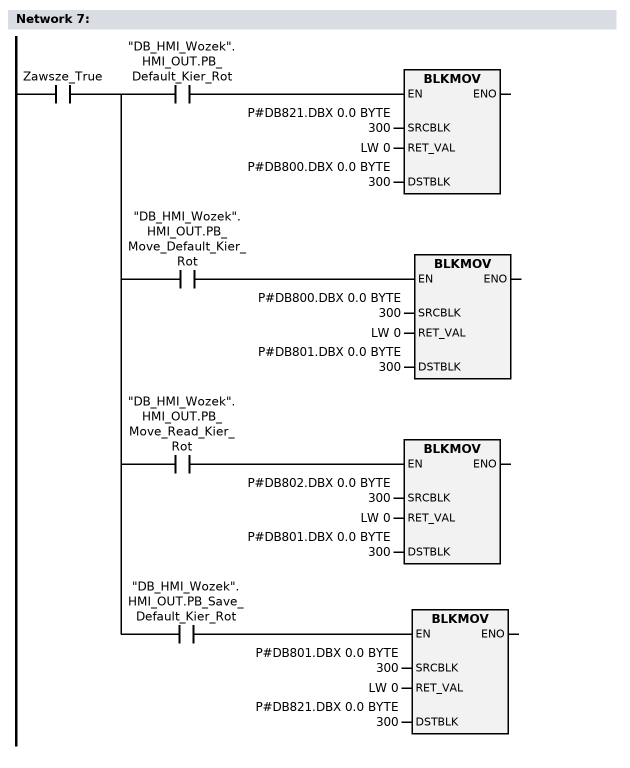
NETWORK
TITLE =
      A     "Zawsze_True";
      =     L 2.0;
      A     L 2.0;
      A     "DB_HMI_Wozek".HMI_OUT.PB_Default_Kier_Rot;
      JNB   _001;
      CALL  "BLKMOV" (
           SRCBLK                   := P#DB821.DBX 0.0 BYTE 300,
           RET_VAL                  := LW 0,
           DSTBLK                   := P#DB800.DBX 0.0 BYTE 300);
_001: NOP   0;
      A     L 2.0;
      A     "DB_HMI_Wozek".HMI_OUT.PB_Move_Default_Kier_Rot;
      JNB   _002;
      CALL  "BLKMOV" (
           SRCBLK                   := P#DB800.DBX 0.0 BYTE 300,
           RET_VAL                  := LW 0,
           DSTBLK                   := P#DB801.DBX 0.0 BYTE 300);
_002: NOP   0;
      A     L 2.0;
      A     "DB_HMI_Wozek".HMI_OUT.PB_Move_Read_Kier_Rot;
      JNB   _003;
      CALL  "BLKMOV" (
           SRCBLK                   := P#DB802.DBX 0.0 BYTE 300,
           RET_VAL                  := LW 0,
           DSTBLK                   := P#DB801.DBX 0.0 BYTE 300);
_003: NOP   0;
      A     L 2.0;
      A     "DB_HMI_Wozek".HMI_OUT.PB_Save_Default_Kier_Rot;
      JNB   _004;
      CALL  "BLKMOV" (
           SRCBLK                   := P#DB801.DBX 0.0 BYTE 300,
           RET_VAL                  := LW 0,
           DSTBLK                   := P#DB821.DBX 0.0 BYTE 300);
_004: NOP   0;
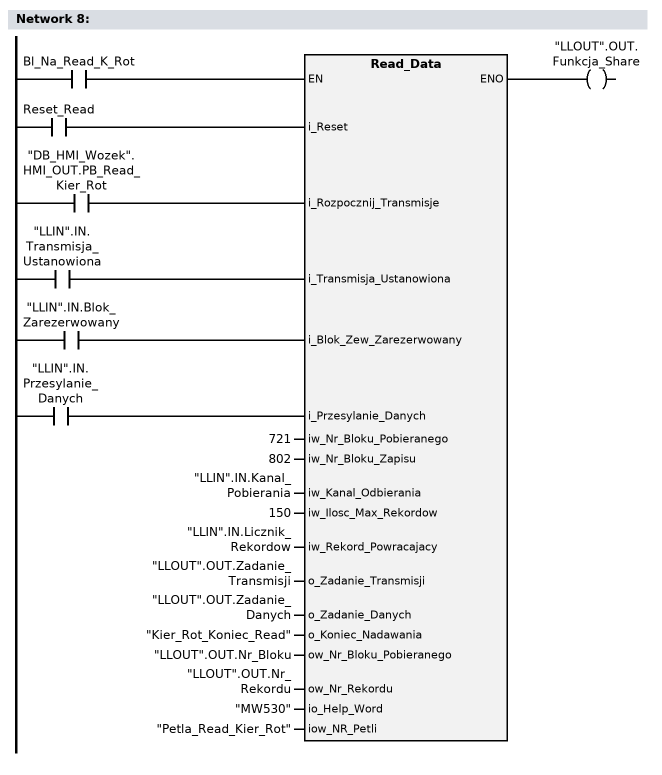
NETWORK
TITLE =
//Funkcja poboru danych
//
      A     "Reset_Read";
      =     L 2.0;
      BLD   103;
      A     "DB_HMI_Wozek".HMI_OUT.PB_Read_Kier_Rot;
      =     L 2.1;
      BLD   103;
      A     "LLIN".IN.Transmisja_Ustanowiona;
      =     L 2.2;
      BLD   103;
      A     "LLIN".IN.Blok_Zarezerwowany;
      =     L 2.3;
      BLD   103;
      A     "LLIN".IN.Przesylanie_Danych;
      =     L 2.4;
      BLD   103;
      A     "Bl_Na_Read_K_Rot";
      JNB   _005;
      CALL  "Read_Data" (
           i_Reset                  := L 2.0,
           i_Rozpocznij_Transmisje  := L 2.1,
           i_Transmisja_Ustanowiona := L 2.2,
           i_Blok_Zew_Zarezerwowany := L 2.3,
           i_Przesylanie_Danych     := L 2.4,
           iw_Nr_Bloku_Pobieranego  := 721,
           iw_Nr_Bloku_Zapisu       := 802,
           iw_Kanal_Odbierania      := "LLIN".IN.Kanal_Pobierania,
           iw_Ilosc_Max_Rekordow    := 150,
           iw_Rekord_Powracajacy    := "LLIN".IN.Licznik_Rekordow,
           o_Zadanie_Transmisji     := "LLOUT".OUT.Zadanie_Transmisji,
           o_Zadanie_Danych         := "LLOUT".OUT.Zadanie_Danych,
           o_Koniec_Nadawania       := "Kier_Rot_Koniec_Read",
           ow_Nr_Bloku_Pobieranego  := "LLOUT".OUT.Nr_Bloku,
           ow_Nr_Rekordu            := "LLOUT".OUT.Nr_Rekordu,
           io_Help_Word             := "MW530",
           iow_NR_Petli             := "Petla_Read_Kier_Rot");
_005: A     BR;
      =     "LLOUT".OUT.Funkcja_Share;
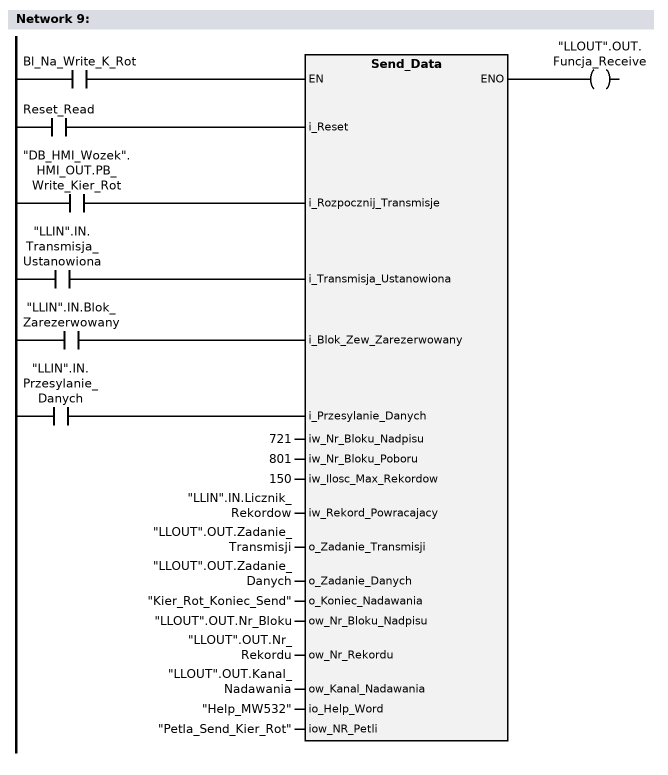
NETWORK
TITLE =
      A     "Reset_Read";
      =     L 2.0;
      BLD   103;
      A     "DB_HMI_Wozek".HMI_OUT.PB_Write_Kier_Rot;
      =     L 2.1;
      BLD   103;
      A     "LLIN".IN.Transmisja_Ustanowiona;
      =     L 2.2;
      BLD   103;
      A     "LLIN".IN.Blok_Zarezerwowany;
      =     L 2.3;
      BLD   103;
      A     "LLIN".IN.Przesylanie_Danych;
      =     L 2.4;
      BLD   103;
      A     "Bl_Na_Write_K_Rot";
      JNB   _006;
      CALL  "Send_Data" (
           i_Reset                  := L 2.0,
           i_Rozpocznij_Transmisje  := L 2.1,
           i_Transmisja_Ustanowiona := L 2.2,
           i_Blok_Zew_Zarezerwowany := L 2.3,
           i_Przesylanie_Danych     := L 2.4,
           iw_Nr_Bloku_Nadpisu      := 721,
           iw_Nr_Bloku_Poboru       := 801,
           iw_Ilosc_Max_Rekordow    := 150,
           iw_Rekord_Powracajacy    := "LLIN".IN.Licznik_Rekordow,
           o_Zadanie_Transmisji     := "LLOUT".OUT.Zadanie_Transmisji,
           o_Zadanie_Danych         := "LLOUT".OUT.Zadanie_Danych,
           o_Koniec_Nadawania       := "Kier_Rot_Koniec_Send",
           ow_Nr_Bloku_Nadpisu      := "LLOUT".OUT.Nr_Bloku,
           ow_Nr_Rekordu            := "LLOUT".OUT.Nr_Rekordu,
           ow_Kanal_Nadawania       := "LLOUT".OUT.Kanal_Nadawania,
           io_Help_Word             := "Help_MW532",
           iow_NR_Petli             := "Petla_Send_Kier_Rot");
_006: A     BR;
      =     "LLOUT".OUT.Funcja_Receive;
END_FUNCTION

FUNCTION "Ekran_Para_Odbieranie" : VOID	// FC 1730
//Ekran para odbieranie marki 505
//
VERSION : 0.1
VAR_INPUT
  Ekran_Aktywny : BOOL ;
  Timmer_Opoz : TIMER ;
END_VAR
VAR_OUTPUT
  Aktywne_Read : BOOL ;
  Aktywne_Write : BOOL ;
  Aktywna_Funkcja : BOOL ;
END_VAR
BEGIN
NETWORK
TITLE =
//Ten network celowo jest wolny
//inputy to i160
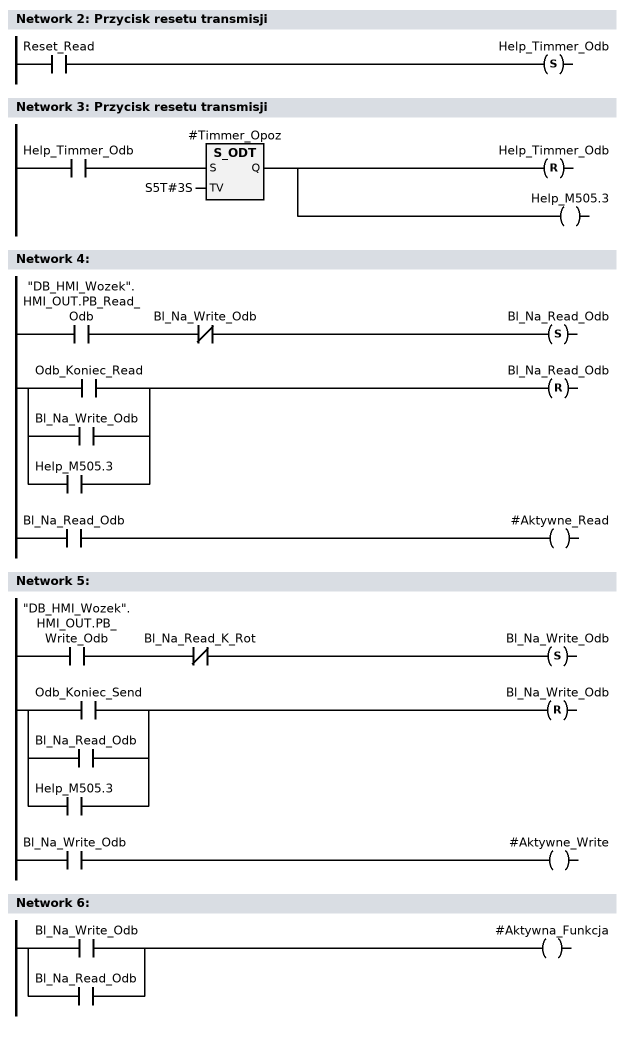
NETWORK
TITLE = Przycisk resetu transmisji
      A     "Reset_Read";
      S     "Help_Timmer_Odb";
NETWORK
TITLE = Przycisk resetu transmisji
      A     "Help_Timmer_Odb";
      L     S5T#3S;
      SD    #Timmer_Opoz;
      NOP   0;
      NOP   0;
      NOP   0;
      A     #Timmer_Opoz;
      R     "Help_Timmer_Odb";
      =     "Help_M505.3";
NETWORK
TITLE =
//Blokada NA Read
      A     "DB_HMI_Wozek".HMI_OUT.PB_Read_Odb;
      AN    "Bl_Na_Write_Odb";
      S     "Bl_Na_Read_Odb";
      A(;
      O     "Odb_Koniec_Read";
      O     "Bl_Na_Write_Odb";
      O     "Help_M505.3";
      );
      R     "Bl_Na_Read_Odb";
      A     "Bl_Na_Read_Odb";
      =     #Aktywne_Read;
NETWORK
TITLE =
//Blokada NA write
      A     "DB_HMI_Wozek".HMI_OUT.PB_Write_Odb;
      AN    "Bl_Na_Read_K_Rot";
      S     "Bl_Na_Write_Odb";
      A(;
      O     "Odb_Koniec_Send";
      O     "Bl_Na_Read_Odb";
      O     "Help_M505.3";
      );
      R     "Bl_Na_Write_Odb";
      A     "Bl_Na_Write_Odb";
      =     #Aktywne_Write;
NETWORK
TITLE =
      O     "Bl_Na_Write_Odb";
      O     "Bl_Na_Read_Odb";
      =     #Aktywna_Funkcja;
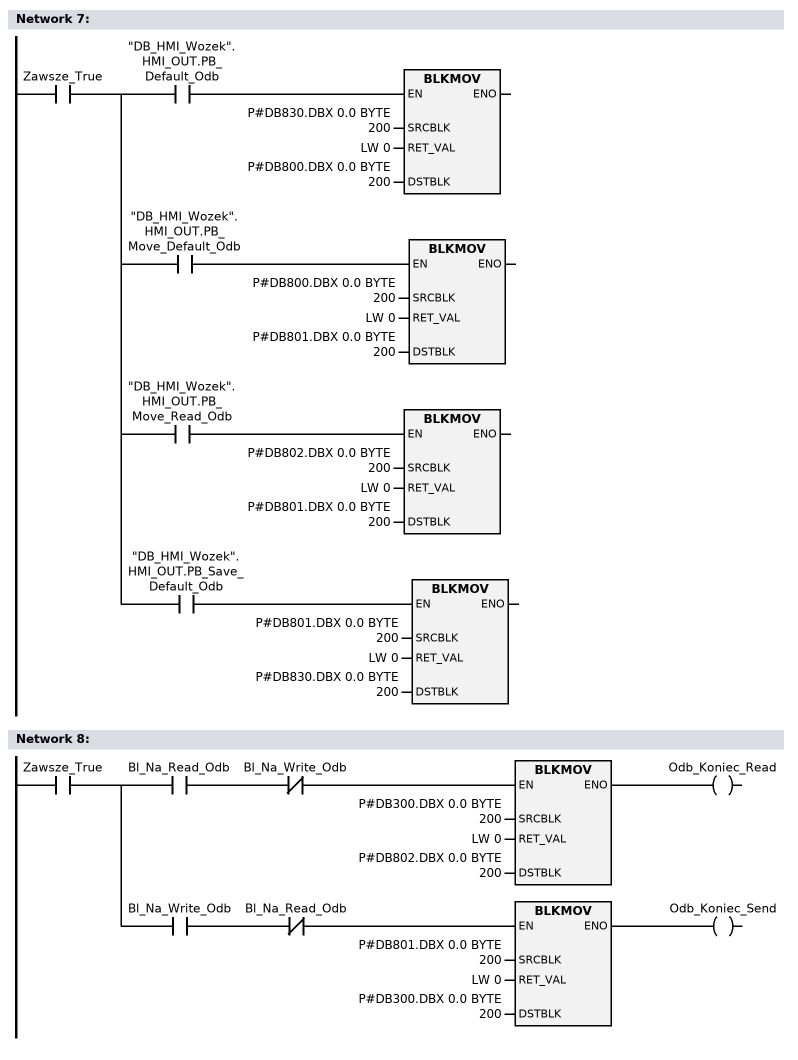
NETWORK
TITLE =
      A     "Zawsze_True";
      =     L 2.0;
      A     L 2.0;
      A     "DB_HMI_Wozek".HMI_OUT.PB_Default_Odb;
      JNB   _001;
      CALL  "BLKMOV" (
           SRCBLK                   := P#DB830.DBX 0.0 BYTE 200,
           RET_VAL                  := LW 0,
           DSTBLK                   := P#DB800.DBX 0.0 BYTE 200);
_001: NOP   0;
      A     L 2.0;
      A     "DB_HMI_Wozek".HMI_OUT.PB_Move_Default_Odb;
      JNB   _002;
      CALL  "BLKMOV" (
           SRCBLK                   := P#DB800.DBX 0.0 BYTE 200,
           RET_VAL                  := LW 0,
           DSTBLK                   := P#DB801.DBX 0.0 BYTE 200);
_002: NOP   0;
      A     L 2.0;
      A     "DB_HMI_Wozek".HMI_OUT.PB_Move_Read_Odb;
      JNB   _003;
      CALL  "BLKMOV" (
           SRCBLK                   := P#DB802.DBX 0.0 BYTE 200,
           RET_VAL                  := LW 0,
           DSTBLK                   := P#DB801.DBX 0.0 BYTE 200);
_003: NOP   0;
      A     L 2.0;
      A     "DB_HMI_Wozek".HMI_OUT.PB_Save_Default_Odb;
      JNB   _004;
      CALL  "BLKMOV" (
           SRCBLK                   := P#DB801.DBX 0.0 BYTE 200,
           RET_VAL                  := LW 0,
           DSTBLK                   := P#DB830.DBX 0.0 BYTE 200);
_004: NOP   0;
NETWORK
TITLE =
//Przesuwanie danych do bloku 300
      A     "Zawsze_True";
      =     L 2.0;
      A     L 2.0;
      A     "Bl_Na_Read_Odb";
      AN    "Bl_Na_Write_Odb";
      JNB   _005;
      CALL  "BLKMOV" (
           SRCBLK                   := P#DB300.DBX 0.0 BYTE 200,
           RET_VAL                  := LW 0,
           DSTBLK                   := P#DB802.DBX 0.0 BYTE 200);
_005: A     BR;
      =     "Odb_Koniec_Read";
      A     L 2.0;
      A     "Bl_Na_Write_Odb";
      AN    "Bl_Na_Read_Odb";
      JNB   _006;
      CALL  "BLKMOV" (
           SRCBLK                   := P#DB801.DBX 0.0 BYTE 200,
           RET_VAL                  := LW 0,
           DSTBLK                   := P#DB300.DBX 0.0 BYTE 200);
_006: A     BR;
      =     "Odb_Koniec_Send";
END_FUNCTION

DATA_BLOCK "Instancja_FB1"	// DB 1
AUTHOR : Kng
VERSION : 0.0
"Stan_Shuttle"
BEGIN
END_DATA_BLOCK

DATA_BLOCK "Instancja_FB3"	// DB 3
AUTHOR : Kng
VERSION : 0.0
"Stanowisko_KB1"
BEGIN
END_DATA_BLOCK

DATA_BLOCK "Instancja_FB4"	// DB 4
AUTHOR : Kng
VERSION : 0.0
"Stanowisko_KB2"
BEGIN
END_DATA_BLOCK

DATA_BLOCK DB 5
VERSION : 0.0
"FB_Uzbrajanie"
BEGIN
END_DATA_BLOCK

DATA_BLOCK DB 6
VERSION : 0.0
"Stan_Intro_Odbieranie"
BEGIN
END_DATA_BLOCK

DATA_BLOCK DB 7
VERSION : 0.0
"Stan_Intro_Pob_I1"
BEGIN
END_DATA_BLOCK

DATA_BLOCK DB 8
AUTHOR : Kng
VERSION : 0.0
"Stan_Intro_Pob_I2"
BEGIN
END_DATA_BLOCK

DATA_BLOCK DB 9
VERSION : 0.0
"Stan_Intro_Pob_I3"
BEGIN
END_DATA_BLOCK

DATA_BLOCK "DB_CONECTOR_KB1"	// DB 11
AUTHOR : Kng
NAME : KB1
VERSION : 0.1
  STRUCT
   Banda_Segbert : UDT 1;	//Adres 1 (Wirtualny)
   Tasma_Obrotnica : UDT 1;	//Adres 2
   Winda : UDT 1;	//Adres 3
   Banda_Wylot_2 : UDT 1;	//Adres 4
   Shuttle : UDT 1;	//Adres 5 (Wirtualny)
   Obrotnica_Pelna : UDT 6;	//Adres 9 (Wirtualny)
   Czujniki_Obr : UDT 7;	//Adres 10
   EStop_Pulpit : UDT 3;	//Adres 20
   Estop_Grzyb_Bezp : UDT 3;	//Adres 21
   Estop_Shuttle : UDT 3;	//ADres 22
  END_STRUCT ;	
BEGIN
   Obrotnica_Pelna.Silnik_OK := TRUE;
END_DATA_BLOCK

DATA_BLOCK "DB_CONECTOR_KB2"	// DB 12
AUTHOR : Kng
NAME : KB2
VERSION : 0.1
  STRUCT
   Banda_Segbert : UDT 1;	//Adres 1 (Wirtualny)
   Tasma_Obrotnica : UDT 1;	//Adres 2
   Winda : UDT 1;	//Adres 3
   Banda_Wylot_2 : UDT 1;	//Adres 4
   Shuttle : UDT 1;	//Adres 5 (Wirtualny)
   Obrotnica_Pelna : UDT 6;	//Adres 9 (Wirtualny)
   Czujniki_Obr : UDT 7;	//Adres 10
   EStop_Pulpit : UDT 3;	//Adres 20
   Estop_Grzyb_Bezp : UDT 3;	//Adres 21
   Estop_Shuttle : UDT 3;	//ADres 22
  END_STRUCT ;	
BEGIN
   Obrotnica_Pelna.Silnik_OK := TRUE;
END_DATA_BLOCK

DATA_BLOCK "DB_CONNECTOR_BUFF"	// DB 13
AUTHOR : Kng
NAME : Buff
VERSION : 0.1
  STRUCT
   Banda_2 : UDT 1;	//Temporary placeholder variable
   Banda_3 : UDT 1;
   Banda_4 : UDT 1;
   Banda_5 : UDT 1;
   Banda_6 : UDT 1;
   Banda_Rez : UDT 1;
   Banda_12 : UDT 1;
   banda_13 : UDT 1;
   Banda_14 : UDT 1;
   Banda_15 : UDT 1;
   Banda_16 : UDT 1;
   Not_Aus_1 : UDT 3;
   Not_Aus_2 : UDT 3;
   Banda_O1_Shuttle : UDT 1;
   Banda_I1_Shuttle : UDT 1;
   Banda_7 : UDT 1;
   Banda_8 : UDT 1;
   Banda_17 : UDT 1;
   Banda_18 : UDT 1;
   Not_Aus_3 : UDT 3;
   Banda_I2_Shuttle : UDT 1;
   Banda_I3_Shuttle : UDT 1;
  END_STRUCT ;	
BEGIN
END_DATA_BLOCK

DATA_BLOCK "DB_CONNECTOR_GEN"	// DB 14
AUTHOR : Kng
NAME : GENDER
VERSION : 0.1
  STRUCT
   Banda_0_Shuttle : UDT 1;	//Adres 1 (Wirtualny)
   Banda_1_Gender : UDT 1;	//Adres 2 (Wirtualny)
  END_STRUCT ;	
BEGIN
END_DATA_BLOCK

DATA_BLOCK "DB_ASI_Prosty_Odczyt_KB1"	// DB 82
AUTHOR : Kng
NAME : KB1
VERSION : 0.1
  STRUCT
   Adres_1_bit_0 : BOOL ;	//Temporary placeholder variable
   Adres_1_bit_1 : BOOL ;
   Adres_1_bit_2 : BOOL ;
   Adres_1_bit_3 : BOOL ;
   Adres_0_bit_0 : BOOL ;	//Temporary placeholder variable
   Adres_0_bit_1 : BOOL ;
   Adres_0_bit_2 : BOOL ;
   Adres_0_bit_3 : BOOL ;
   Adres_3_bit_0 : BOOL ;	//Temporary placeholder variable
   Adres_3_bit_1 : BOOL ;
   Adres_3_bit_2 : BOOL ;
   Adres_3_bit_3 : BOOL ;
   Adres_2_bit_0 : BOOL ;	//Temporary placeholder variable
   Adres_2_bit_1 : BOOL ;
   Adres_2_bit_2 : BOOL ;
   Adres_2_bit_3 : BOOL ;
   Adres_5_bit_0 : BOOL ;	//Temporary placeholder variable
   Adres_5_bit_1 : BOOL ;
   Adres_5_bit_2 : BOOL ;
   Adres_5_bit_3 : BOOL ;
   Adres_4_bit_0 : BOOL ;	//Temporary placeholder variable
   Adres_4_bit_1 : BOOL ;
   Adres_4_bit_2 : BOOL ;
   Adres_4_bit_3 : BOOL ;
   Adres_7_bit_0 : BOOL ;	//Temporary placeholder variable
   Adres_7_bit_1 : BOOL ;
   Adres_7_bit_2 : BOOL ;
   Adres_7_bit_3 : BOOL ;
   Adres_6_bit_0 : BOOL ;	//Temporary placeholder variable
   Adres_6_bit_1 : BOOL ;
   Adres_6_bit_2 : BOOL ;
   Adres_6_bit_3 : BOOL ;
   Adres_9_bit_0 : BOOL ;	//Temporary placeholder variable
   Adres_9_bit_1 : BOOL ;
   Adres_9_bit_2 : BOOL ;
   Adres_9_bit_3 : BOOL ;
   Adres_8_bit_0 : BOOL ;	//Temporary placeholder variable
   Adres_8_bit_1 : BOOL ;
   Adres_8_bit_2 : BOOL ;
   Adres_8_bit_3 : BOOL ;
   Adres_11_bit_0 : BOOL ;	//Temporary placeholder variable
   Adres_11_bit_1 : BOOL ;
   Adres_11_bit_2 : BOOL ;
   Adres_11_bit_3 : BOOL ;
   Adres_10_bit_0 : BOOL ;	//Temporary placeholder variable
   Adres_10_bit_1 : BOOL ;
   Adres_10_bit_2 : BOOL ;
   Adres_10_bit_3 : BOOL ;
   Adres_13_bit_0 : BOOL ;	//Temporary placeholder variable
   Adres_13_bit_1 : BOOL ;
   Adres_13_bit_2 : BOOL ;
   Adres_13_bit_3 : BOOL ;
   Adres_12_bit_0 : BOOL ;	//Temporary placeholder variable
   Adres_12_bit_1 : BOOL ;
   Adres_12_bit_2 : BOOL ;
   Adres_12_bit_3 : BOOL ;
   Adres_15_bit_0 : BOOL ;	//Temporary placeholder variable
   Adres_15_bit_1 : BOOL ;
   Adres_15_bit_2 : BOOL ;
   Adres_15_bit_3 : BOOL ;
   Adres_14_bit_0 : BOOL ;	//Temporary placeholder variable
   Adres_14_bit_1 : BOOL ;
   Adres_14_bit_2 : BOOL ;
   Adres_14_bit_3 : BOOL ;
   Adres_17_bit_0 : BOOL ;	//Temporary placeholder variable
   Adres_17_bit_1 : BOOL ;
   Adres_17_bit_2 : BOOL ;
   Adres_17_bit_3 : BOOL ;
   Adres_16_bit_0 : BOOL ;	//Temporary placeholder variable
   Adres_16_bit_1 : BOOL ;
   Adres_16_bit_2 : BOOL ;
   Adres_16_bit_3 : BOOL ;
   Adres_19_bit_0 : BOOL ;	//Temporary placeholder variable
   Adres_19_bit_1 : BOOL ;
   Adres_19_bit_2 : BOOL ;
   Adres_19_bit_3 : BOOL ;
   Adres_18_bit_0 : BOOL ;	//Temporary placeholder variable
   Adres_18_bit_1 : BOOL ;
   Adres_18_bit_2 : BOOL ;
   Adres_18_bit_3 : BOOL ;
   Adres_21_bit_0 : BOOL ;	//Temporary placeholder variable
   Adres_21_bit_1 : BOOL ;
   Adres_21_bit_2 : BOOL ;
   Adres_21_bit_3 : BOOL ;
   Adres_20_bit_0 : BOOL ;	//Temporary placeholder variable
   Adres_20_bit_1 : BOOL ;
   Adres_20_bit_2 : BOOL ;
   Adres_20_bit_3 : BOOL ;
   Adres_23_bit_0 : BOOL ;	//Temporary placeholder variable
   Adres_23_bit_1 : BOOL ;
   Adres_23_bit_2 : BOOL ;
   Adres_23_bit_3 : BOOL ;
   Adres_22_bit_0 : BOOL ;	//Temporary placeholder variable
   Adres_22_bit_1 : BOOL ;
   Adres_22_bit_2 : BOOL ;
   Adres_22_bit_3 : BOOL ;
   Adres_25_bit_0 : BOOL ;	//Temporary placeholder variable
   Adres_25_bit_1 : BOOL ;
   Adres_25_bit_2 : BOOL ;
   Adres_25_bit_3 : BOOL ;
   Adres_24_bit_0 : BOOL ;	//Temporary placeholder variable
   Adres_24_bit_1 : BOOL ;
   Adres_24_bit_2 : BOOL ;
   Adres_24_bit_3 : BOOL ;
   Adres_27_bit_0 : BOOL ;	//Temporary placeholder variable
   Adres_27_bit_1 : BOOL ;
   Adres_27_bit_2 : BOOL ;
   Adres_27_bit_3 : BOOL ;
   Adres_26_bit_0 : BOOL ;	//Temporary placeholder variable
   Adres_26_bit_1 : BOOL ;
   Adres_26_bit_2 : BOOL ;
   Adres_26_bit_3 : BOOL ;
   Adres_29_bit_0 : BOOL ;	//Temporary placeholder variable
   Adres_29_bit_1 : BOOL ;
   Adres_29_bit_2 : BOOL ;
   Adres_29_bit_3 : BOOL ;
   Adres_28_bit_0 : BOOL ;	//Temporary placeholder variable
   Adres_28_bit_1 : BOOL ;
   Adres_28_bit_2 : BOOL ;
   Adres_28_bit_3 : BOOL ;
   Adres_31_bit_0 : BOOL ;	//Temporary placeholder variable
   Adres_31_bit_1 : BOOL ;
   Adres_31_bit_2 : BOOL ;
   Adres_31_bit_3 : BOOL ;
   Adres_30_bit_0 : BOOL ;	//Temporary placeholder variable
   Adres_30_bit_1 : BOOL ;
   Adres_30_bit_2 : BOOL ;
   Adres_30_bit_3 : BOOL ;
  END_STRUCT ;	
BEGIN
END_DATA_BLOCK

DATA_BLOCK "DB_ASI_Prosty_Zapis_KB1"	// DB 83
AUTHOR : Kng
NAME : KB1
VERSION : 0.1
  STRUCT
   Adres_1_bit_0 : BOOL ;	//Temporary placeholder variable
   Adres_1_bit_1 : BOOL ;
   Adres_1_bit_2 : BOOL ;
   Adres_1_bit_3 : BOOL ;
   Adres_0_bit_0 : BOOL ;	//Temporary placeholder variable
   Adres_0_bit_1 : BOOL ;
   Adres_0_bit_2 : BOOL ;
   Adres_0_bit_3 : BOOL ;
   Adres_3_bit_0 : BOOL ;	//Temporary placeholder variable
   Adres_3_bit_1 : BOOL ;
   Adres_3_bit_2 : BOOL ;
   Adres_3_bit_3 : BOOL ;
   Adres_2_bit_0 : BOOL ;	//Temporary placeholder variable
   Adres_2_bit_1 : BOOL ;
   Adres_2_bit_2 : BOOL ;
   Adres_2_bit_3 : BOOL ;
   Adres_5_bit_0 : BOOL ;	//Temporary placeholder variable
   Adres_5_bit_1 : BOOL ;
   Adres_5_bit_2 : BOOL ;
   Adres_5_bit_3 : BOOL ;
   Adres_4_bit_0 : BOOL ;	//Temporary placeholder variable
   Adres_4_bit_1 : BOOL ;
   Adres_4_bit_2 : BOOL ;
   Adres_4_bit_3 : BOOL ;
   Adres_7_bit_0 : BOOL ;	//Temporary placeholder variable
   Adres_7_bit_1 : BOOL ;
   Adres_7_bit_2 : BOOL ;
   Adres_7_bit_3 : BOOL ;
   Adres_6_bit_0 : BOOL ;	//Temporary placeholder variable
   Adres_6_bit_1 : BOOL ;
   Adres_6_bit_2 : BOOL ;
   Adres_6_bit_3 : BOOL ;
   Adres_9_bit_0 : BOOL ;	//Temporary placeholder variable
   Adres_9_bit_1 : BOOL ;
   Adres_9_bit_2 : BOOL ;
   Adres_9_bit_3 : BOOL ;
   Adres_8_bit_0 : BOOL ;	//Temporary placeholder variable
   Adres_8_bit_1 : BOOL ;
   Adres_8_bit_2 : BOOL ;
   Adres_8_bit_3 : BOOL ;
   Adres_11_bit_0 : BOOL ;	//Temporary placeholder variable
   Adres_11_bit_1 : BOOL ;
   Adres_11_bit_2 : BOOL ;
   Adres_11_bit_3 : BOOL ;
   Adres_10_bit_0 : BOOL ;	//Temporary placeholder variable
   Adres_10_bit_1 : BOOL ;
   Adres_10_bit_2 : BOOL ;
   Adres_10_bit_3 : BOOL ;
   Adres_13_bit_0 : BOOL ;	//Temporary placeholder variable
   Adres_13_bit_1 : BOOL ;
   Adres_13_bit_2 : BOOL ;
   Adres_13_bit_3 : BOOL ;
   Adres_12_bit_0 : BOOL ;	//Temporary placeholder variable
   Adres_12_bit_1 : BOOL ;
   Adres_12_bit_2 : BOOL ;
   Adres_12_bit_3 : BOOL ;
   Adres_15_bit_0 : BOOL ;	//Temporary placeholder variable
   Adres_15_bit_1 : BOOL ;
   Adres_15_bit_2 : BOOL ;
   Adres_15_bit_3 : BOOL ;
   Adres_14_bit_0 : BOOL ;	//Temporary placeholder variable
   Adres_14_bit_1 : BOOL ;
   Adres_14_bit_2 : BOOL ;
   Adres_14_bit_3 : BOOL ;
   Adres_17_bit_0 : BOOL ;	//Temporary placeholder variable
   Adres_17_bit_1 : BOOL ;
   Adres_17_bit_2 : BOOL ;
   Adres_17_bit_3 : BOOL ;
   Adres_16_bit_0 : BOOL ;	//Temporary placeholder variable
   Adres_16_bit_1 : BOOL ;
   Adres_16_bit_2 : BOOL ;
   Adres_16_bit_3 : BOOL ;
   Adres_19_bit_0 : BOOL ;	//Temporary placeholder variable
   Adres_19_bit_1 : BOOL ;
   Adres_19_bit_2 : BOOL ;
   Adres_19_bit_3 : BOOL ;
   Adres_18_bit_0 : BOOL ;	//Temporary placeholder variable
   Adres_18_bit_1 : BOOL ;
   Adres_18_bit_2 : BOOL ;
   Adres_18_bit_3 : BOOL ;
   Adres_21_bit_0 : BOOL ;	//Temporary placeholder variable
   Adres_21_bit_1 : BOOL ;
   Adres_21_bit_2 : BOOL ;
   Adres_21_bit_3 : BOOL ;
   Adres_20_bit_0 : BOOL ;	//Temporary placeholder variable
   Adres_20_bit_1 : BOOL ;
   Adres_20_bit_2 : BOOL ;
   Adres_20_bit_3 : BOOL ;
   Adres_23_bit_0 : BOOL ;	//Temporary placeholder variable
   Adres_23_bit_1 : BOOL ;
   Adres_23_bit_2 : BOOL ;
   Adres_23_bit_3 : BOOL ;
   Adres_22_bit_0 : BOOL ;	//Temporary placeholder variable
   Adres_22_bit_1 : BOOL ;
   Adres_22_bit_2 : BOOL ;
   Adres_22_bit_3 : BOOL ;
   Adres_25_bit_0 : BOOL ;	//Temporary placeholder variable
   Adres_25_bit_1 : BOOL ;
   Adres_25_bit_2 : BOOL ;
   Adres_25_bit_3 : BOOL ;
   Adres_24_bit_0 : BOOL ;	//Temporary placeholder variable
   Adres_24_bit_1 : BOOL ;
   Adres_24_bit_2 : BOOL ;
   Adres_24_bit_3 : BOOL ;
   Adres_27_bit_0 : BOOL ;	//Temporary placeholder variable
   Adres_27_bit_1 : BOOL ;
   Adres_27_bit_2 : BOOL ;
   Adres_27_bit_3 : BOOL ;
   Adres_26_bit_0 : BOOL ;	//Temporary placeholder variable
   Adres_26_bit_1 : BOOL ;
   Adres_26_bit_2 : BOOL ;
   Adres_26_bit_3 : BOOL ;
   Adres_29_bit_0 : BOOL ;	//Temporary placeholder variable
   Adres_29_bit_1 : BOOL ;
   Adres_29_bit_2 : BOOL ;
   Adres_29_bit_3 : BOOL ;
   Adres_28_bit_0 : BOOL ;	//Temporary placeholder variable
   Adres_28_bit_1 : BOOL ;
   Adres_28_bit_2 : BOOL ;
   Adres_28_bit_3 : BOOL ;
   Adres_31_bit_0 : BOOL ;	//Temporary placeholder variable
   Adres_31_bit_1 : BOOL ;
   Adres_31_bit_2 : BOOL ;
   Adres_31_bit_3 : BOOL ;
   Adres_30_bit_0 : BOOL ;	//Temporary placeholder variable
   Adres_30_bit_1 : BOOL ;
   Adres_30_bit_2 : BOOL ;
   Adres_30_bit_3 : BOOL ;
  END_STRUCT ;	
BEGIN
END_DATA_BLOCK

DATA_BLOCK "DB_ASI_Prosty_Odczyt_KB2"	// DB 84
AUTHOR : Kng
NAME : KB2
VERSION : 0.1
  STRUCT
   Adres_1_bit_0 : BOOL ;	//Temporary placeholder variable
   Adres_1_bit_1 : BOOL ;
   Adres_1_bit_2 : BOOL ;
   Adres_1_bit_3 : BOOL ;
   Adres_0_bit_0 : BOOL ;	//Temporary placeholder variable
   Adres_0_bit_1 : BOOL ;
   Adres_0_bit_2 : BOOL ;
   Adres_0_bit_3 : BOOL ;
   Adres_3_bit_0 : BOOL ;	//Temporary placeholder variable
   Adres_3_bit_1 : BOOL ;
   Adres_3_bit_2 : BOOL ;
   Adres_3_bit_3 : BOOL ;
   Adres_2_bit_0 : BOOL ;	//Temporary placeholder variable
   Adres_2_bit_1 : BOOL ;
   Adres_2_bit_2 : BOOL ;
   Adres_2_bit_3 : BOOL ;
   Adres_5_bit_0 : BOOL ;	//Temporary placeholder variable
   Adres_5_bit_1 : BOOL ;
   Adres_5_bit_2 : BOOL ;
   Adres_5_bit_3 : BOOL ;
   Adres_4_bit_0 : BOOL ;	//Temporary placeholder variable
   Adres_4_bit_1 : BOOL ;
   Adres_4_bit_2 : BOOL ;
   Adres_4_bit_3 : BOOL ;
   Adres_7_bit_0 : BOOL ;	//Temporary placeholder variable
   Adres_7_bit_1 : BOOL ;
   Adres_7_bit_2 : BOOL ;
   Adres_7_bit_3 : BOOL ;
   Adres_6_bit_0 : BOOL ;	//Temporary placeholder variable
   Adres_6_bit_1 : BOOL ;
   Adres_6_bit_2 : BOOL ;
   Adres_6_bit_3 : BOOL ;
   Adres_9_bit_0 : BOOL ;	//Temporary placeholder variable
   Adres_9_bit_1 : BOOL ;
   Adres_9_bit_2 : BOOL ;
   Adres_9_bit_3 : BOOL ;
   Adres_8_bit_0 : BOOL ;	//Temporary placeholder variable
   Adres_8_bit_1 : BOOL ;
   Adres_8_bit_2 : BOOL ;
   Adres_8_bit_3 : BOOL ;
   Adres_11_bit_0 : BOOL ;	//Temporary placeholder variable
   Adres_11_bit_1 : BOOL ;
   Adres_11_bit_2 : BOOL ;
   Adres_11_bit_3 : BOOL ;
   Adres_10_bit_0 : BOOL ;	//Temporary placeholder variable
   Adres_10_bit_1 : BOOL ;
   Adres_10_bit_2 : BOOL ;
   Adres_10_bit_3 : BOOL ;
   Adres_13_bit_0 : BOOL ;	//Temporary placeholder variable
   Adres_13_bit_1 : BOOL ;
   Adres_13_bit_2 : BOOL ;
   Adres_13_bit_3 : BOOL ;
   Adres_12_bit_0 : BOOL ;	//Temporary placeholder variable
   Adres_12_bit_1 : BOOL ;
   Adres_12_bit_2 : BOOL ;
   Adres_12_bit_3 : BOOL ;
   Adres_15_bit_0 : BOOL ;	//Temporary placeholder variable
   Adres_15_bit_1 : BOOL ;
   Adres_15_bit_2 : BOOL ;
   Adres_15_bit_3 : BOOL ;
   Adres_14_bit_0 : BOOL ;	//Temporary placeholder variable
   Adres_14_bit_1 : BOOL ;
   Adres_14_bit_2 : BOOL ;
   Adres_14_bit_3 : BOOL ;
   Adres_17_bit_0 : BOOL ;	//Temporary placeholder variable
   Adres_17_bit_1 : BOOL ;
   Adres_17_bit_2 : BOOL ;
   Adres_17_bit_3 : BOOL ;
   Adres_16_bit_0 : BOOL ;	//Temporary placeholder variable
   Adres_16_bit_1 : BOOL ;
   Adres_16_bit_2 : BOOL ;
   Adres_16_bit_3 : BOOL ;
   Adres_19_bit_0 : BOOL ;	//Temporary placeholder variable
   Adres_19_bit_1 : BOOL ;
   Adres_19_bit_2 : BOOL ;
   Adres_19_bit_3 : BOOL ;
   Adres_18_bit_0 : BOOL ;	//Temporary placeholder variable
   Adres_18_bit_1 : BOOL ;
   Adres_18_bit_2 : BOOL ;
   Adres_18_bit_3 : BOOL ;
   Adres_21_bit_0 : BOOL ;	//Temporary placeholder variable
   Adres_21_bit_1 : BOOL ;
   Adres_21_bit_2 : BOOL ;
   Adres_21_bit_3 : BOOL ;
   Adres_20_bit_0 : BOOL ;	//Temporary placeholder variable
   Adres_20_bit_1 : BOOL ;
   Adres_20_bit_2 : BOOL ;
   Adres_20_bit_3 : BOOL ;
   Adres_23_bit_0 : BOOL ;	//Temporary placeholder variable
   Adres_23_bit_1 : BOOL ;
   Adres_23_bit_2 : BOOL ;
   Adres_23_bit_3 : BOOL ;
   Adres_22_bit_0 : BOOL ;	//Temporary placeholder variable
   Adres_22_bit_1 : BOOL ;
   Adres_22_bit_2 : BOOL ;
   Adres_22_bit_3 : BOOL ;
   Adres_25_bit_0 : BOOL ;	//Temporary placeholder variable
   Adres_25_bit_1 : BOOL ;
   Adres_25_bit_2 : BOOL ;
   Adres_25_bit_3 : BOOL ;
   Adres_24_bit_0 : BOOL ;	//Temporary placeholder variable
   Adres_24_bit_1 : BOOL ;
   Adres_24_bit_2 : BOOL ;
   Adres_24_bit_3 : BOOL ;
   Adres_27_bit_0 : BOOL ;	//Temporary placeholder variable
   Adres_27_bit_1 : BOOL ;
   Adres_27_bit_2 : BOOL ;
   Adres_27_bit_3 : BOOL ;
   Adres_26_bit_0 : BOOL ;	//Temporary placeholder variable
   Adres_26_bit_1 : BOOL ;
   Adres_26_bit_2 : BOOL ;
   Adres_26_bit_3 : BOOL ;
   Adres_29_bit_0 : BOOL ;	//Temporary placeholder variable
   Adres_29_bit_1 : BOOL ;
   Adres_29_bit_2 : BOOL ;
   Adres_29_bit_3 : BOOL ;
   Adres_28_bit_0 : BOOL ;	//Temporary placeholder variable
   Adres_28_bit_1 : BOOL ;
   Adres_28_bit_2 : BOOL ;
   Adres_28_bit_3 : BOOL ;
   Adres_31_bit_0 : BOOL ;	//Temporary placeholder variable
   Adres_31_bit_1 : BOOL ;
   Adres_31_bit_2 : BOOL ;
   Adres_31_bit_3 : BOOL ;
   Adres_30_bit_0 : BOOL ;	//Temporary placeholder variable
   Adres_30_bit_1 : BOOL ;
   Adres_30_bit_2 : BOOL ;
   Adres_30_bit_3 : BOOL ;
  END_STRUCT ;	
BEGIN
END_DATA_BLOCK

DATA_BLOCK "DB_ASi_Prosty_Zapis_KB2"	// DB 85
AUTHOR : Kng
NAME : KB2
VERSION : 0.1
  STRUCT
   Adres_1_bit_0 : BOOL ;	//Temporary placeholder variable
   Adres_1_bit_1 : BOOL ;
   Adres_1_bit_2 : BOOL ;
   Adres_1_bit_3 : BOOL ;
   Adres_0_bit_0 : BOOL ;	//Temporary placeholder variable
   Adres_0_bit_1 : BOOL ;
   Adres_0_bit_2 : BOOL ;
   Adres_0_bit_3 : BOOL ;
   Adres_3_bit_0 : BOOL ;	//Temporary placeholder variable
   Adres_3_bit_1 : BOOL ;
   Adres_3_bit_2 : BOOL ;
   Adres_3_bit_3 : BOOL ;
   Adres_2_bit_0 : BOOL ;	//Temporary placeholder variable
   Adres_2_bit_1 : BOOL ;
   Adres_2_bit_2 : BOOL ;
   Adres_2_bit_3 : BOOL ;
   Adres_5_bit_0 : BOOL ;	//Temporary placeholder variable
   Adres_5_bit_1 : BOOL ;
   Adres_5_bit_2 : BOOL ;
   Adres_5_bit_3 : BOOL ;
   Adres_4_bit_0 : BOOL ;	//Temporary placeholder variable
   Adres_4_bit_1 : BOOL ;
   Adres_4_bit_2 : BOOL ;
   Adres_4_bit_3 : BOOL ;
   Adres_7_bit_0 : BOOL ;	//Temporary placeholder variable
   Adres_7_bit_1 : BOOL ;
   Adres_7_bit_2 : BOOL ;
   Adres_7_bit_3 : BOOL ;
   Adres_6_bit_0 : BOOL ;	//Temporary placeholder variable
   Adres_6_bit_1 : BOOL ;
   Adres_6_bit_2 : BOOL ;
   Adres_6_bit_3 : BOOL ;
   Adres_9_bit_0 : BOOL ;	//Temporary placeholder variable
   Adres_9_bit_1 : BOOL ;
   Adres_9_bit_2 : BOOL ;
   Adres_9_bit_3 : BOOL ;
   Adres_8_bit_0 : BOOL ;	//Temporary placeholder variable
   Adres_8_bit_1 : BOOL ;
   Adres_8_bit_2 : BOOL ;
   Adres_8_bit_3 : BOOL ;
   Adres_11_bit_0 : BOOL ;	//Temporary placeholder variable
   Adres_11_bit_1 : BOOL ;
   Adres_11_bit_2 : BOOL ;
   Adres_11_bit_3 : BOOL ;
   Adres_10_bit_0 : BOOL ;	//Temporary placeholder variable
   Adres_10_bit_1 : BOOL ;
   Adres_10_bit_2 : BOOL ;
   Adres_10_bit_3 : BOOL ;
   Adres_13_bit_0 : BOOL ;	//Temporary placeholder variable
   Adres_13_bit_1 : BOOL ;
   Adres_13_bit_2 : BOOL ;
   Adres_13_bit_3 : BOOL ;
   Adres_12_bit_0 : BOOL ;	//Temporary placeholder variable
   Adres_12_bit_1 : BOOL ;
   Adres_12_bit_2 : BOOL ;
   Adres_12_bit_3 : BOOL ;
   Adres_15_bit_0 : BOOL ;	//Temporary placeholder variable
   Adres_15_bit_1 : BOOL ;
   Adres_15_bit_2 : BOOL ;
   Adres_15_bit_3 : BOOL ;
   Adres_14_bit_0 : BOOL ;	//Temporary placeholder variable
   Adres_14_bit_1 : BOOL ;
   Adres_14_bit_2 : BOOL ;
   Adres_14_bit_3 : BOOL ;
   Adres_17_bit_0 : BOOL ;	//Temporary placeholder variable
   Adres_17_bit_1 : BOOL ;
   Adres_17_bit_2 : BOOL ;
   Adres_17_bit_3 : BOOL ;
   Adres_16_bit_0 : BOOL ;	//Temporary placeholder variable
   Adres_16_bit_1 : BOOL ;
   Adres_16_bit_2 : BOOL ;
   Adres_16_bit_3 : BOOL ;
   Adres_19_bit_0 : BOOL ;	//Temporary placeholder variable
   Adres_19_bit_1 : BOOL ;
   Adres_19_bit_2 : BOOL ;
   Adres_19_bit_3 : BOOL ;
   Adres_18_bit_0 : BOOL ;	//Temporary placeholder variable
   Adres_18_bit_1 : BOOL ;
   Adres_18_bit_2 : BOOL ;
   Adres_18_bit_3 : BOOL ;
   Adres_21_bit_0 : BOOL ;	//Temporary placeholder variable
   Adres_21_bit_1 : BOOL ;
   Adres_21_bit_2 : BOOL ;
   Adres_21_bit_3 : BOOL ;
   Adres_20_bit_0 : BOOL ;	//Temporary placeholder variable
   Adres_20_bit_1 : BOOL ;
   Adres_20_bit_2 : BOOL ;
   Adres_20_bit_3 : BOOL ;
   Adres_23_bit_0 : BOOL ;	//Temporary placeholder variable
   Adres_23_bit_1 : BOOL ;
   Adres_23_bit_2 : BOOL ;
   Adres_23_bit_3 : BOOL ;
   Adres_22_bit_0 : BOOL ;	//Temporary placeholder variable
   Adres_22_bit_1 : BOOL ;
   Adres_22_bit_2 : BOOL ;
   Adres_22_bit_3 : BOOL ;
   Adres_25_bit_0 : BOOL ;	//Temporary placeholder variable
   Adres_25_bit_1 : BOOL ;
   Adres_25_bit_2 : BOOL ;
   Adres_25_bit_3 : BOOL ;
   Adres_24_bit_0 : BOOL ;	//Temporary placeholder variable
   Adres_24_bit_1 : BOOL ;
   Adres_24_bit_2 : BOOL ;
   Adres_24_bit_3 : BOOL ;
   Adres_27_bit_0 : BOOL ;	//Temporary placeholder variable
   Adres_27_bit_1 : BOOL ;
   Adres_27_bit_2 : BOOL ;
   Adres_27_bit_3 : BOOL ;
   Adres_26_bit_0 : BOOL ;	//Temporary placeholder variable
   Adres_26_bit_1 : BOOL ;
   Adres_26_bit_2 : BOOL ;
   Adres_26_bit_3 : BOOL ;
   Adres_29_bit_0 : BOOL ;	//Temporary placeholder variable
   Adres_29_bit_1 : BOOL ;
   Adres_29_bit_2 : BOOL ;
   Adres_29_bit_3 : BOOL ;
   Adres_28_bit_0 : BOOL ;	//Temporary placeholder variable
   Adres_28_bit_1 : BOOL ;
   Adres_28_bit_2 : BOOL ;
   Adres_28_bit_3 : BOOL ;
   Adres_31_bit_0 : BOOL ;	//Temporary placeholder variable
   Adres_31_bit_1 : BOOL ;
   Adres_31_bit_2 : BOOL ;
   Adres_31_bit_3 : BOOL ;
   Adres_30_bit_0 : BOOL ;	//Temporary placeholder variable
   Adres_30_bit_1 : BOOL ;
   Adres_30_bit_2 : BOOL ;
   Adres_30_bit_3 : BOOL ;
  END_STRUCT ;	
BEGIN
END_DATA_BLOCK

DATA_BLOCK "DB_ASi_Prosty_Odczyt_Buf"	// DB 86
AUTHOR : Kng
NAME : Buff
VERSION : 0.1
  STRUCT
   Adres_1_bit_0 : BOOL ;	//Temporary placeholder variable
   Adres_1_bit_1 : BOOL ;
   Adres_1_bit_2 : BOOL ;
   Adres_1_bit_3 : BOOL ;
   Adres_0_bit_0 : BOOL ;	//Temporary placeholder variable
   Adres_0_bit_1 : BOOL ;
   Adres_0_bit_2 : BOOL ;
   Adres_0_bit_3 : BOOL ;
   Adres_3_bit_0 : BOOL ;	//Temporary placeholder variable
   Adres_3_bit_1 : BOOL ;
   Adres_3_bit_2 : BOOL ;
   Adres_3_bit_3 : BOOL ;
   Adres_2_bit_0 : BOOL ;	//Temporary placeholder variable
   Adres_2_bit_1 : BOOL ;
   Adres_2_bit_2 : BOOL ;
   Adres_2_bit_3 : BOOL ;
   Adres_5_bit_0 : BOOL ;	//Temporary placeholder variable
   Adres_5_bit_1 : BOOL ;
   Adres_5_bit_2 : BOOL ;
   Adres_5_bit_3 : BOOL ;
   Adres_4_bit_0 : BOOL ;	//Temporary placeholder variable
   Adres_4_bit_1 : BOOL ;
   Adres_4_bit_2 : BOOL ;
   Adres_4_bit_3 : BOOL ;
   Adres_7_bit_0 : BOOL ;	//Temporary placeholder variable
   Adres_7_bit_1 : BOOL ;
   Adres_7_bit_2 : BOOL ;
   Adres_7_bit_3 : BOOL ;
   Adres_6_bit_0 : BOOL ;	//Temporary placeholder variable
   Adres_6_bit_1 : BOOL ;
   Adres_6_bit_2 : BOOL ;
   Adres_6_bit_3 : BOOL ;
   Adres_9_bit_0 : BOOL ;	//Temporary placeholder variable
   Adres_9_bit_1 : BOOL ;
   Adres_9_bit_2 : BOOL ;
   Adres_9_bit_3 : BOOL ;
   Adres_8_bit_0 : BOOL ;	//Temporary placeholder variable
   Adres_8_bit_1 : BOOL ;
   Adres_8_bit_2 : BOOL ;
   Adres_8_bit_3 : BOOL ;
   Adres_11_bit_0 : BOOL ;	//Temporary placeholder variable
   Adres_11_bit_1 : BOOL ;
   Adres_11_bit_2 : BOOL ;
   Adres_11_bit_3 : BOOL ;
   Adres_10_bit_0 : BOOL ;	//Temporary placeholder variable
   Adres_10_bit_1 : BOOL ;
   Adres_10_bit_2 : BOOL ;
   Adres_10_bit_3 : BOOL ;
   Adres_13_bit_0 : BOOL ;	//Temporary placeholder variable
   Adres_13_bit_1 : BOOL ;
   Adres_13_bit_2 : BOOL ;
   Adres_13_bit_3 : BOOL ;
   Adres_12_bit_0 : BOOL ;	//Temporary placeholder variable
   Adres_12_bit_1 : BOOL ;
   Adres_12_bit_2 : BOOL ;
   Adres_12_bit_3 : BOOL ;
   Adres_15_bit_0 : BOOL ;	//Temporary placeholder variable
   Adres_15_bit_1 : BOOL ;
   Adres_15_bit_2 : BOOL ;
   Adres_15_bit_3 : BOOL ;
   Adres_14_bit_0 : BOOL ;	//Temporary placeholder variable
   Adres_14_bit_1 : BOOL ;
   Adres_14_bit_2 : BOOL ;
   Adres_14_bit_3 : BOOL ;
   Adres_17_bit_0 : BOOL ;	//Temporary placeholder variable
   Adres_17_bit_1 : BOOL ;
   Adres_17_bit_2 : BOOL ;
   Adres_17_bit_3 : BOOL ;
   Adres_16_bit_0 : BOOL ;	//Temporary placeholder variable
   Adres_16_bit_1 : BOOL ;
   Adres_16_bit_2 : BOOL ;
   Adres_16_bit_3 : BOOL ;
   Adres_19_bit_0 : BOOL ;	//Temporary placeholder variable
   Adres_19_bit_1 : BOOL ;
   Adres_19_bit_2 : BOOL ;
   Adres_19_bit_3 : BOOL ;
   Adres_18_bit_0 : BOOL ;	//Temporary placeholder variable
   Adres_18_bit_1 : BOOL ;
   Adres_18_bit_2 : BOOL ;
   Adres_18_bit_3 : BOOL ;
   Adres_21_bit_0 : BOOL ;	//Temporary placeholder variable
   Adres_21_bit_1 : BOOL ;
   Adres_21_bit_2 : BOOL ;
   Adres_21_bit_3 : BOOL ;
   Adres_20_bit_0 : BOOL ;	//Temporary placeholder variable
   Adres_20_bit_1 : BOOL ;
   Adres_20_bit_2 : BOOL ;
   Adres_20_bit_3 : BOOL ;
   Adres_23_bit_0 : BOOL ;	//Temporary placeholder variable
   Adres_23_bit_1 : BOOL ;
   Adres_23_bit_2 : BOOL ;
   Adres_23_bit_3 : BOOL ;
   Adres_22_bit_0 : BOOL ;	//Temporary placeholder variable
   Adres_22_bit_1 : BOOL ;
   Adres_22_bit_2 : BOOL ;
   Adres_22_bit_3 : BOOL ;
   Adres_25_bit_0 : BOOL ;	//Temporary placeholder variable
   Adres_25_bit_1 : BOOL ;
   Adres_25_bit_2 : BOOL ;
   Adres_25_bit_3 : BOOL ;
   Adres_24_bit_0 : BOOL ;	//Temporary placeholder variable
   Adres_24_bit_1 : BOOL ;
   Adres_24_bit_2 : BOOL ;
   Adres_24_bit_3 : BOOL ;
   Adres_27_bit_0 : BOOL ;	//Temporary placeholder variable
   Adres_27_bit_1 : BOOL ;
   Adres_27_bit_2 : BOOL ;
   Adres_27_bit_3 : BOOL ;
   Adres_26_bit_0 : BOOL ;	//Temporary placeholder variable
   Adres_26_bit_1 : BOOL ;
   Adres_26_bit_2 : BOOL ;
   Adres_26_bit_3 : BOOL ;
   Adres_29_bit_0 : BOOL ;	//Temporary placeholder variable
   Adres_29_bit_1 : BOOL ;
   Adres_29_bit_2 : BOOL ;
   Adres_29_bit_3 : BOOL ;
   Adres_28_bit_0 : BOOL ;	//Temporary placeholder variable
   Adres_28_bit_1 : BOOL ;
   Adres_28_bit_2 : BOOL ;
   Adres_28_bit_3 : BOOL ;
   Adres_31_bit_0 : BOOL ;	//Temporary placeholder variable
   Adres_31_bit_1 : BOOL ;
   Adres_31_bit_2 : BOOL ;
   Adres_31_bit_3 : BOOL ;
   Adres_30_bit_0 : BOOL ;	//Temporary placeholder variable
   Adres_30_bit_1 : BOOL ;
   Adres_30_bit_2 : BOOL ;
   Adres_30_bit_3 : BOOL ;
  END_STRUCT ;	
BEGIN
END_DATA_BLOCK

DATA_BLOCK "DB_ASi_Prosty_Zapis_Buf"	// DB 87
AUTHOR : Kng
NAME : Buff
VERSION : 0.1
  STRUCT
   Adres_1_bit_0 : BOOL ;	//Temporary placeholder variable
   Adres_1_bit_1 : BOOL ;
   Adres_1_bit_2 : BOOL ;
   Adres_1_bit_3 : BOOL ;
   Adres_0_bit_0 : BOOL ;	//Temporary placeholder variable
   Adres_0_bit_1 : BOOL ;
   Adres_0_bit_2 : BOOL ;
   Adres_0_bit_3 : BOOL ;
   Adres_3_bit_0 : BOOL ;	//Temporary placeholder variable
   Adres_3_bit_1 : BOOL ;
   Adres_3_bit_2 : BOOL ;
   Adres_3_bit_3 : BOOL ;
   Adres_2_bit_0 : BOOL ;	//Temporary placeholder variable
   Adres_2_bit_1 : BOOL ;
   Adres_2_bit_2 : BOOL ;
   Adres_2_bit_3 : BOOL ;
   Adres_5_bit_0 : BOOL ;	//Temporary placeholder variable
   Adres_5_bit_1 : BOOL ;
   Adres_5_bit_2 : BOOL ;
   Adres_5_bit_3 : BOOL ;
   Adres_4_bit_0 : BOOL ;	//Temporary placeholder variable
   Adres_4_bit_1 : BOOL ;
   Adres_4_bit_2 : BOOL ;
   Adres_4_bit_3 : BOOL ;
   Adres_7_bit_0 : BOOL ;	//Temporary placeholder variable
   Adres_7_bit_1 : BOOL ;
   Adres_7_bit_2 : BOOL ;
   Adres_7_bit_3 : BOOL ;
   Adres_6_bit_0 : BOOL ;	//Temporary placeholder variable
   Adres_6_bit_1 : BOOL ;
   Adres_6_bit_2 : BOOL ;
   Adres_6_bit_3 : BOOL ;
   Adres_9_bit_0 : BOOL ;	//Temporary placeholder variable
   Adres_9_bit_1 : BOOL ;
   Adres_9_bit_2 : BOOL ;
   Adres_9_bit_3 : BOOL ;
   Adres_8_bit_0 : BOOL ;	//Temporary placeholder variable
   Adres_8_bit_1 : BOOL ;
   Adres_8_bit_2 : BOOL ;
   Adres_8_bit_3 : BOOL ;
   Adres_11_bit_0 : BOOL ;	//Temporary placeholder variable
   Adres_11_bit_1 : BOOL ;
   Adres_11_bit_2 : BOOL ;
   Adres_11_bit_3 : BOOL ;
   Adres_10_bit_0 : BOOL ;	//Temporary placeholder variable
   Adres_10_bit_1 : BOOL ;
   Adres_10_bit_2 : BOOL ;
   Adres_10_bit_3 : BOOL ;
   Adres_13_bit_0 : BOOL ;	//Temporary placeholder variable
   Adres_13_bit_1 : BOOL ;
   Adres_13_bit_2 : BOOL ;
   Adres_13_bit_3 : BOOL ;
   Adres_12_bit_0 : BOOL ;	//Temporary placeholder variable
   Adres_12_bit_1 : BOOL ;
   Adres_12_bit_2 : BOOL ;
   Adres_12_bit_3 : BOOL ;
   Adres_15_bit_0 : BOOL ;	//Temporary placeholder variable
   Adres_15_bit_1 : BOOL ;
   Adres_15_bit_2 : BOOL ;
   Adres_15_bit_3 : BOOL ;
   Adres_14_bit_0 : BOOL ;	//Temporary placeholder variable
   Adres_14_bit_1 : BOOL ;
   Adres_14_bit_2 : BOOL ;
   Adres_14_bit_3 : BOOL ;
   Adres_17_bit_0 : BOOL ;	//Temporary placeholder variable
   Adres_17_bit_1 : BOOL ;
   Adres_17_bit_2 : BOOL ;
   Adres_17_bit_3 : BOOL ;
   Adres_16_bit_0 : BOOL ;	//Temporary placeholder variable
   Adres_16_bit_1 : BOOL ;
   Adres_16_bit_2 : BOOL ;
   Adres_16_bit_3 : BOOL ;
   Adres_19_bit_0 : BOOL ;	//Temporary placeholder variable
   Adres_19_bit_1 : BOOL ;
   Adres_19_bit_2 : BOOL ;
   Adres_19_bit_3 : BOOL ;
   Adres_18_bit_0 : BOOL ;	//Temporary placeholder variable
   Adres_18_bit_1 : BOOL ;
   Adres_18_bit_2 : BOOL ;
   Adres_18_bit_3 : BOOL ;
   Adres_21_bit_0 : BOOL ;	//Temporary placeholder variable
   Adres_21_bit_1 : BOOL ;
   Adres_21_bit_2 : BOOL ;
   Adres_21_bit_3 : BOOL ;
   Adres_20_bit_0 : BOOL ;	//Temporary placeholder variable
   Adres_20_bit_1 : BOOL ;
   Adres_20_bit_2 : BOOL ;
   Adres_20_bit_3 : BOOL ;
   Adres_23_bit_0 : BOOL ;	//Temporary placeholder variable
   Adres_23_bit_1 : BOOL ;
   Adres_23_bit_2 : BOOL ;
   Adres_23_bit_3 : BOOL ;
   Adres_22_bit_0 : BOOL ;	//Temporary placeholder variable
   Adres_22_bit_1 : BOOL ;
   Adres_22_bit_2 : BOOL ;
   Adres_22_bit_3 : BOOL ;
   Adres_25_bit_0 : BOOL ;	//Temporary placeholder variable
   Adres_25_bit_1 : BOOL ;
   Adres_25_bit_2 : BOOL ;
   Adres_25_bit_3 : BOOL ;
   Adres_24_bit_0 : BOOL ;	//Temporary placeholder variable
   Adres_24_bit_1 : BOOL ;
   Adres_24_bit_2 : BOOL ;
   Adres_24_bit_3 : BOOL ;
   Adres_27_bit_0 : BOOL ;	//Temporary placeholder variable
   Adres_27_bit_1 : BOOL ;
   Adres_27_bit_2 : BOOL ;
   Adres_27_bit_3 : BOOL ;
   Adres_26_bit_0 : BOOL ;	//Temporary placeholder variable
   Adres_26_bit_1 : BOOL ;
   Adres_26_bit_2 : BOOL ;
   Adres_26_bit_3 : BOOL ;
   Adres_29_bit_0 : BOOL ;	//Temporary placeholder variable
   Adres_29_bit_1 : BOOL ;
   Adres_29_bit_2 : BOOL ;
   Adres_29_bit_3 : BOOL ;
   Adres_28_bit_0 : BOOL ;	//Temporary placeholder variable
   Adres_28_bit_1 : BOOL ;
   Adres_28_bit_2 : BOOL ;
   Adres_28_bit_3 : BOOL ;
   Adres_31_bit_0 : BOOL ;	//Temporary placeholder variable
   Adres_31_bit_1 : BOOL ;
   Adres_31_bit_2 : BOOL ;
   Adres_31_bit_3 : BOOL ;
   Adres_30_bit_0 : BOOL ;	//Temporary placeholder variable
   Adres_30_bit_1 : BOOL ;
   Adres_30_bit_2 : BOOL ;
   Adres_30_bit_3 : BOOL ;
  END_STRUCT ;	
BEGIN
END_DATA_BLOCK

DATA_BLOCK "Bledy_Shuttle"	// DB 116
VERSION : 0.1
  STRUCT
   Bledy : STRUCT
    Przek_Bezp_Nie_Ok : BOOL ;	//Blad przekanika bezpieczenstwa [I4.1 s. 10]
    Blad_Kom_Odbieranie : BOOL ;	//Blad komunikacji z odbieraniem [FC119]
    Bezpieczniki_Nie_Ok : BOOL ;	//Wyzwolenie wylacznika termicznego [I4.0 s. 10]
    Mayser_Nie_Ok : BOOL ;	//Wyzwolenie listwy bezpieczenstwa [I4.2 s.10]
    Foto_Zle_Pokrycie : BOOL ;	//Niedozwolone pokrycie fotokomorek obecnosci palety [I5.2,I5.3 s.11]
    Hamulec_Reczny_Rewizja : BOOL ;	//Hamulec reczny odbezpieczony [I5.6 s 11]
    Skaner_Wym_Przod_Reset : BOOL ;	//Skaner przod wymagany reset [I6.1 s.12]
    Skaner_Przod_Error : BOOL ;	//Blad Skanera przedniego lub jego  zabrudzenie [I6.2 s.12]
    Skaner_Przod_Strefa : BOOL ;	//Skaner przedni strefa wyzwolona I[I6.3 s.12]
    Skaner_Wym_Tyl_Reset : BOOL ;	//Skaner tylni wymagany reset [I7.1 s.12]
    Skaner_Tyl_Error : BOOL ;	//Blad Skanera tylniego lub jego  zabrudzenie [I7.2 s.12]
    Skaner_Tyl_Strefa : BOOL ;	//Skaner tylni strefa wyzwolona [I7.3 s.12]
    Obwody_Zew_Nie_Ok : BOOL ;	//Obwody bezpieczenstwa zewnetrzne nie Ok [I8.1 s.14](Not-Aus Slupy)
    Falownik_Sew_Blad : BOOL ;	//Blad falownika SEW [FC101]
    Falownik_Sew_N_Ready : BOOL ;	//Falownik sew nie gotowy [FC101]
    Falownik_Lenze_Blad : BOOL ;	//Blad falownika Lenze [FC101]
    Warunki_Startu_N_OK : BOOL ;	//Warunki startu Sew nie spelnione [FC101]
    Blad_Zwolnienia : BOOL ;	//Blad zwolnienia tasmy transportera [FC30]
    Help_int : INT ;	//Rezerwa dla booli
    Nr_Bledu_Sew : INT ;	//Blad specyficzny sew do odczytania
    Prad_Aktualny : INT ;	//Prad aktualny SEW [FC101]
    Predkosc_Aktualna : INT ;	//Predkosc akutualna wozka [FC101]
    Reserwa_Int : INT ;
    REserwa_Int1 : INT ;
   END_STRUCT ;
  END_STRUCT ;	
BEGIN
END_DATA_BLOCK

DATA_BLOCK "Bledy_KB1"	// DB 117
VERSION : 0.1
  STRUCT
   Obwod_Bezp_1_Nie_OK : BOOL ;	//Przekaznik bezpieczenstwa stanowisko nie ok [I24.0-KB2]{I14.0-KB1] s.12
   Obwod_Bezp_2_Nie_OK : BOOL ;	//Przekaznik bezpieczenstwa wozek nie ok [I24.1-KB2][I14.1-KB1] s.12
   Petla_Bezp_Nie_Ok : BOOL ;	//Petla bezpiecznikow nie OK [I24.2-KB2][I14.2-KB1] s.12
   Blad_Silnika_Rolki_Obr : BOOL ;	//Blad silnika rolek obrotnica Adres 2 s.32
   Blad_Silnika_Rolki_Winda : BOOL ;	//Blad silnika rolek winda Adres 3 s.33
   Blad_Silnika_Rolki_Wy_2 : BOOL ;	//Blad silnika rolek wylot 2 Adres 4 s.34
   Blad_Silnika_Obrotu : BOOL ;	//Blad falownika Lenze obronicy Adres DP [8-KB2][4-KB1] s.35
   Blad_Not_Aus_Pulpit : BOOL ;	//Przycisk Not-Aus pulpit sterowniczy Adres 20 s.40
   Blad_Not_Aus_Grzyb_Obr : BOOL ;	//Blad Not-Aus grzyb obrotnica Adres 21 s.40
   Blad_Not_Aus_Wozek : BOOL ;	//Blad Not-Aus na s³upie od wozka Adres 22 s.40
  END_STRUCT ;	
BEGIN
END_DATA_BLOCK

DATA_BLOCK "Bledy_KB2"	// DB 118
VERSION : 0.1
  STRUCT
   Obwod_Bezp_1_Nie_OK : BOOL ;	//Przekaznik bezpieczenstwa stanowisko nie ok [I24.0-KB2]{I14.0-KB1] s.12
   Obwod_Bezp_2_Nie_OK : BOOL ;	//Przekaznik bezpieczenstwa wozek nie ok [I24.1-KB2][I14.1-KB1] s.12
   Petla_Bezp_Nie_Ok : BOOL ;	//Petla bezpiecznikow nie OK [I24.2-KB2][I14.2-KB1] s.12
   Blad_Silnika_Rolki_Obr : BOOL ;	//Blad silnika rolek obrotnica Adres 2 s.32
   Blad_Silnika_Rolki_Winda : BOOL ;	//Blad silnika rolek winda Adres 3 s.33
   Blad_Silnika_Rolki_Wy_2 : BOOL ;	//Blad silnika rolek wylot 2 Adres 4 s.34
   Blad_Silnika_Obrotu : BOOL ;	//Blad falownika Lenze obronicy Adres DP [8-KB2][4-KB1] s.35
   Blad_Not_Aus_Pulpit : BOOL ;	//Przycisk Not-Aus pulpit sterowniczy Adres 20 s.40
   Blad_Not_Aus_Grzyb_Obr : BOOL ;	//Blad Not-Aus grzyb obrotnica Adres 21 s.40
   Blad_Not_Aus_Wozek : BOOL ;	//Blad Not-Aus na s³upie od wozka Adres 22 s.40
  END_STRUCT ;	
BEGIN
END_DATA_BLOCK

DATA_BLOCK "Bledy_Buffor"	// DB 119
VERSION : 0.1
  STRUCT
   Blad_Silnik_Banda_2 : BOOL ;	//Blad silnika Adres 2 - bandy odbieranie
   Blad_Silnik_Banda_3 : BOOL ;	//Blad silnika Adres 3 - bandy odbieranie
   Blad_Silnik_Banda_4 : BOOL ;	//Blad silnika Adres 4 - bandy odbieranie
   Blad_Silnik_Banda_5 : BOOL ;	//Blad silnika Adres 5 - bandy odbieranie
   Blad_Silnik_Banda_6 : BOOL ;	//Blad silnika Adres 6 - bandy odbieranie
   Blad_Silnik_Banda_Rez : BOOL ;
   Blad_Silnik_Banda_12 : BOOL ;	//Blad silnika Adres 12 - bandy pobieranie
   Blad_Silnik_Banda_13 : BOOL ;	//Blad silnika Adres 13 - bandy pobieranie
   Blad_Silnik_Banda_14 : BOOL ;	//Blad silnika Adres 14 - bandy pobieranie
   Blad_Silnik_Banda_15 : BOOL ;	//Blad silnika Adres 15 - bandy pobieranie
   Blad_Silnik_Banda_16 : BOOL ;	//Blad silnika Adres 16 - bandy pobieranie
   Blad_Not_Aus_Pulpit : BOOL ;	//Blad Not-Aus pulpit Adres 20
   Blad_Not_Aus_KB1 : BOOL ;	//Blad Not-Aus na slupie Kolbus 1 (Adres 22) s.9
   Blad_Not_Aus_KB2 : BOOL ;	//Blad Not-Aus na slupie Kolbus 2 (Adres 22) s.9
   Blad_Not_Aus_Slupy : BOOL ;	//Blad Not-Aus na ktoryms slupie  (Adres 22)
   Blad_Not_Aus_Buff : BOOL ;	//Blad Not-Aus na slupie Buffory  (Adres 23)
   Przekaznik_Bezp_1_Nie_Ok : BOOL ;	//Przekaznik Bezpieczenstwa Pulpit Nie OK [I10.0] s.12
   Przekaznik_Bezp_2_Nie_Ok : BOOL ;	//Przekanik Bezpieczenstwa od Wozka Nie OK [I10.1] s.12
   Blad_Wozka_Widl : BOOL ;	//Wozek przyslania fotokomorke [I8.7] s.10
   Napiecie_Shuttle_Wyl : BOOL ;	//Napiecie na szynoprzewod nie za³¹czone [Q8.3] s.18
   Blad_Silnik_Banda_7 : BOOL ;	//Blad silnika Adres 7- bandy pobieranie
   Blad_Silnik_Banda_17 : BOOL ;	//Blad silnika Adres 17 - bandy pobieranie
   Blad_Silnik_Banda_8 : BOOL ;	//Blad silnika Adres 8 - bandy pobieranie
   Blad_Silnik_Banda_18 : BOOL ;	//Blad silnika Adres 18 - bandy pobieranie
   Blad_Not_Aus_Pulpit_2 : BOOL ;	//Blad Not-Aus pulpit Adres 24
  END_STRUCT ;	
BEGIN
END_DATA_BLOCK

DATA_BLOCK "DB_HMI_KB1"	// DB 121
AUTHOR : Kng
NAME : HMI_KB2
VERSION : 0.1
  STRUCT
   HMI_IN : STRUCT 	//Zmienne wchodzace do HMI nie nadpisywane W HMI (100 bajtow)
    Reserwa_in : BOOL ;
    Winda_W_Dole : BOOL ;	//Winda w dole dbx0.1
    Winda_W_Gorze : BOOL ;	//Winda w gorze
    Zawor_Winda : BOOL ;
    Silnik_Winda : BOOL ;
    Foto_Winda_Przod : BOOL ;
    Foto_Winda_Tyl : BOOL ;
    Silnik_Banda_Winda_OK : BOOL ;
    Obrot_Pozycja_Na_Winde : BOOL ;
    Obrot_Pozycja_Na_Wylot_2 : BOOL ;
    Foto_Obrotnica_Przod : BOOL ;
    Foto_Obrotnica_Tyl : BOOL ;
    Silnik_Banda_Obrot_OK : BOOL ;
    Silnik_Obrot_OK : BOOL ;
    Foto_Wozek_Przod : BOOL ;
    Foto_Wozek_Tyl : BOOL ;
    Silnik_Wozek_OK : BOOL ;
    Foto_Segbert_Przod : BOOL ;
    Foto_Segbert_Tyl : BOOL ;
    Segbert_Strefa_Ok : BOOL ;
    Segbert_Silnik_Ok : BOOL ;
    Foto_Wylot_2_Przod : BOOL ;
    Foto_Wylot_2_Tyl : BOOL ;
    Wylot_2_Silnik_OK : BOOL ;
    Not_Aus_Pulpit_Ok : BOOL ;
    Not_Aus_Slupek_OK : BOOL ;
    Not_Aus_Wozek_OK : BOOL ;
    Uzbrajanie_Aktywne : BOOL ;	//dbx3.3
    Uzbrajanie_Kier_Lewo : BOOL ;
    Uzbrajanie_Kier_Prawo : BOOL ;
    Zasprzeglenie_KB1 : BOOL ;
    Rezerwa_113 : BOOL ;
    Silnik_Segbert_CW : BOOL ;
    Wybor_Kier_Spedycja : BOOL ;	//dbx4.1
    Wybor_Kier_Intro : BOOL ;
    Wybor_Wiazanie_Pop : BOOL ;
    Wybor_Wiazanie_Wzdl : BOOL ;
    Wybor_Deklowanie : BOOL ;
    Wybor_Foliowanie : BOOL ;
    Silnik_Segbert_CCW : BOOL ;
    Silnik_Obrot_Banda_CCW : BOOL ;
    Silnik_Obrot_Banda_CW : BOOL ;
    Silnik_Winda_CCW : BOOL ;
    Silnik_Winda_CW : BOOL ;
    Silnik_Wylot2_CCW : BOOL ;
    Silnik_Wylot2_CW : BOOL ;
    Silnik_Wozek_CCW : BOOL ;
    Silnik_Wozek_CW : BOOL ;
    Silnik_Segbert_Praca : BOOL ;
    Silnik_Obrot_Banda_Praca : BOOL ;
    Silnik_Winda_Praca : BOOL ;
    Silnik_Wylot2_Praca : BOOL ;
    Silnik_Wozek_Praca : BOOL ;
    Silnik_Obrotnica_CCW : BOOL ;
    Silnik_Obrotnica_CW : BOOL ;
    Obrotnica_Na_Winde : BYTE ;
    Obrotnica_Na_Wylot2 : BYTE ;
    Ruch_Banda_Segbert : BYTE ;
    Ruch_Banda_Obrotnicy : BYTE ;
    Ruch_Banda_Winda : BYTE ;
    Ruch_Banda_Wozek : BYTE ;
    Ruch_Banda_Wylot2 : BYTE ;
    Status_B_Segbert_uzbr : BOOL ;
    Status_B_Segbert_foliow : BOOL ;
    Status_B_Segbert_deklow : BOOL ;
    Status_B_Segbert_W_wzdl : BOOL ;
    Status_B_Segbert_W_poprz : BOOL ;
    Status_B_Segbert_widoczn : BOOL ;
    res : BOOL ;
    res1 : BOOL ;
    Status_B_Obr_0st_uzbr : BOOL ;
    Status_B_Obr_0st_foliow : BOOL ;
    Status_B_Obr_0st_deklow : BOOL ;
    Status_B_Obr_0st_W_wzdl : BOOL ;
    Status_B_Obr_0st_W_poprz : BOOL ;
    Status_B_Obr_0st_widoczn : BOOL ;
    res2 : BOOL ;
    res3 : BOOL ;
    Status_B_Winda_uzbr : BOOL ;
    Status_B_Winda_foliow : BOOL ;
    Status_B_Winda_deklow : BOOL ;
    Status_B_Winda_W_wzdl : BOOL ;
    Status_B_Winda_W_poprz : BOOL ;
    Status_B_Winda_widoczn : BOOL ;
    res10 : BOOL ;
    res11 : BOOL ;
    Status_B_Wozek_uzbr : BOOL ;
    Status_B_Wozek_foliow : BOOL ;
    Status_B_Wozek_deklow : BOOL ;
    Status_B_Wozek_W_wzdl : BOOL ;
    Status_B_Wozek_W_poprz : BOOL ;
    Status_B_Wozek_widoczn : BOOL ;
    res4 : BOOL ;
    res5 : BOOL ;
    Status_B_Wylot2_uzbr : BOOL ;
    Status_B_Wylot2_foliow : BOOL ;
    Status_B_Wylot2_deklow : BOOL ;
    Status_B_Wylot2_W_wzdl : BOOL ;
    Status_B_Wylot2_W_poprz : BOOL ;
    Status_B_Wylot2_widoczn : BOOL ;
    res6 : BOOL ;
    res7 : BOOL ;
    Status_B_Obr_90st_uzbr : BOOL ;
    Status_B_Obr_90st_foliow : BOOL ;
    Status_B_Obr_90st_deklow : BOOL ;
    Status_B_Obr_90st_W_wzdl : BOOL ;
    Status_B_Obr_90st_W_popr : BOOL ;
    Status_B_Obr_90st_widocz : BOOL ;
    res8 : BOOL ;
    res9 : BOOL ;
    Winda_Dol : BOOL ;
    Winda_Srodek_Dol : BOOL ;
    Winda_Srodek_Gora : BOOL ;
    Winda_Gora : BOOL ;
    Paleta_Winda_Inf_KB1 : DINT ;
    Paleta_Ruch_Pion : INT ;
    Paleta_Ruch_Poziom : INT ;
    Paleta_Winda_Inf_KB1_HMI : DINT ;
    Tablica_IN_INT : ARRAY  [1 .. 13 ] OF INT ;
    Tablica_IN_DWORD : ARRAY  [1 .. 8 ] OF DINT ;
    Aktualna_Data : DATE_AND_TIME ;
   END_STRUCT ;
   HMI_OUT : STRUCT 	//Zmienne wychodzace z HMI Nie nadpisywane w sterowniku od 100 bajta
    Tryb_Uzbrajania_Palety : BOOL ;	//Paleta bedzie uzbrajana dbx100.0
    Tryb_Pracy_Inline : BOOL ;	//Kierunek wylotu palety 1-winda 0-bok dbx100.1
    Ladunek_Na_Intro : BOOL ;
    Reserwa_11 : BOOL ;
    Reserwa_12 : BOOL ;
    Reset_Bledow : BOOL ;	//Reset bledow maszyny
    Reserwa_14 : BOOL ;
    Reserwa_15 : BOOL ;
    Reserwa_16 : BOOL ;
    Reserwa_17 : BOOL ;
    Reserwa_18 : BOOL ;
    Reserwa_19 : BOOL ;
    Reserwa_110 : BOOL ;
    Reserwa_111 : BOOL ;
    Reserwa_112 : BOOL ;
    Reserwa_113 : BOOL ;
    Wybrano_Kier_Spedycje : BOOL ;	//Jedzie na Gender ( dbx2.0)
    Wybrano_Kier_Intro : BOOL ;	//Jedzie na bandy buffory
    Wybrano_Wiaz_Pop : BOOL ;
    Wybrano_Wiaz_Wzdlu : BOOL ;	//Wybrano wiazanie wzdluzne
    Wybrano_Deklowanie : BOOL ;	//wybrano deklowanie
    Wybrano_Foliowanie : BOOL ;
    Kier_Spedycja_Aktywny : BOOL ;
    Kierunek_Intro_Aktywny : BOOL ;
    Wiazanie_Pop_Aktywne : BOOL ;
    Wiazanie_Wzdl_Aktywne : BOOL ;
    Deklowanie_Aktywne : BOOL ;
    Foliowanie_Aktywne : BOOL ;
    reserwa : BOOL ;
    reserwa1 : BOOL ;
    reserwa2 : BOOL ;
    reserwa3 : BOOL ;
    reserwa4 : INT ;	//Wartosc % predkosci z ladunkiem
    Predkosc_Cargo : INT ;	//Wartosc % predkosci z ladunkiem
    Tablica_OUT_INT : ARRAY  [1 .. 21 ] OF INT ;
    Maska_Zadania : INT ;
    Tablica_OUT_DWORD : ARRAY  [1 .. 9 ] OF DWORD ;
    Reserwa_DWORD : DWORD ;
    Aktualna_Data : DATE_AND_TIME ;
   END_STRUCT ;
   HMI_IN_OUT : STRUCT 	//Zmienne nadpisywane w sterowniku i w HMI od 200 bajta
    Reserwa_in_out : BOOL ;
    io_Reserwa : INT ;	//Rodzaj wybranego wlotu
    Predkosc_Obrotnicy : DINT  := L#20;	//dbd4
    Tablica_IN_OUT_INT : ARRAY  [1 .. 22 ] OF INT ;
    Tablica_IN_OUT_DWORD : ARRAY  [1 .. 10 ] OF DWORD ;
    Aktualna_Data : DATE_AND_TIME ;
   END_STRUCT ;
  END_STRUCT ;	
BEGIN
   HMI_IN_OUT.Predkosc_Obrotnicy := L#20;
END_DATA_BLOCK

DATA_BLOCK "DB_HMI_KB2"	// DB 122
AUTHOR : Kng
NAME : HMI_KB2
VERSION : 0.1
  STRUCT
   HMI_IN : STRUCT 	//Zmienne wchodzace do HMI nie nadpisywane W HMI (100 bajtow)
    Reserwa_in : BOOL ;
    Winda_W_Dole : BOOL ;	//Winda w dole dbx0.1
    Winda_W_Gorze : BOOL ;	//Winda w gorze
    Zawor_Winda : BOOL ;
    Silnik_Winda : BOOL ;
    Foto_Winda_Przod : BOOL ;
    Foto_Winda_Tyl : BOOL ;
    Silnik_Banda_Winda_OK : BOOL ;
    Obrot_Pozycja_Na_Winde : BOOL ;
    Obrot_Pozycja_Na_Wylot_2 : BOOL ;
    Foto_Obrotnica_Przod : BOOL ;
    Foto_Obrotnica_Tyl : BOOL ;
    Silnik_Banda_Obrot_OK : BOOL ;
    Silnik_Obrot_OK : BOOL ;
    Foto_Wozek_Przod : BOOL ;
    Foto_Wozek_Tyl : BOOL ;
    Silnik_Wozek_OK : BOOL ;
    Foto_Segbert_Przod : BOOL ;
    Foto_Segbert_Tyl : BOOL ;
    Segbert_Strefa_Ok : BOOL ;
    Segbert_Silnik_Ok : BOOL ;
    Foto_Wylot_2_Przod : BOOL ;
    Foto_Wylot_2_Tyl : BOOL ;
    Wylot_2_Silnik_OK : BOOL ;
    Not_Aus_Pulpit_Ok : BOOL ;
    Not_Aus_Slupek_OK : BOOL ;
    Not_Aus_Wozek_OK : BOOL ;
    Uzbrajanie_Aktywne : BOOL ;	//dbx3.3
    Uzbrajanie_Kier_Lewo : BOOL ;
    Uzbrajanie_Kier_Prawo : BOOL ;
    Zasprzeglenie_KB2 : BOOL ;
    Rezerwa_113 : BOOL ;
    Silnik_Segbert_CW : BOOL ;
    Wybor_Kier_Spedycja : BOOL ;	//dbx4.1
    Wybor_Kier_Intro : BOOL ;
    Wybor_Wiazanie_Pop : BOOL ;
    Wybor_Wiazanie_Wzdl : BOOL ;
    Wybor_Deklowanie : BOOL ;
    Wybor_Foliowanie : BOOL ;
    Silnik_Segbert_CCW : BOOL ;
    Silnik_Obrot_Banda_CCW : BOOL ;
    Silnik_Obrot_Banda_CW : BOOL ;
    Silnik_Winda_CCW : BOOL ;
    Silnik_Winda_CW : BOOL ;
    Silnik_Wylot2_CCW : BOOL ;
    Silnik_Wylot2_CW : BOOL ;
    Silnik_Wozek_CCW : BOOL ;
    Silnik_Wozek_CW : BOOL ;
    Silnik_Segbert_Praca : BOOL ;
    Silnik_Obrot_Banda_Praca : BOOL ;
    Silnik_Winda_Praca : BOOL ;
    Silnik_Wylot2_Praca : BOOL ;
    Silnik_Wozek_Praca : BOOL ;
    Silnik_Obrotnica_CCW : BOOL ;
    Silnik_Obrotnica_CW : BOOL ;
    Obrotnica_Na_Winde : BYTE ;
    Obrotnica_Na_Wylot2 : BYTE ;
    Ruch_Banda_Segbert : BYTE ;
    Ruch_Banda_Obrotnicy : BYTE ;
    Ruch_Banda_Winda : BYTE ;
    Ruch_Banda_Wozek : BYTE ;
    Ruch_Banda_Wylot2 : BYTE ;
    Status_B_Segbert_uzbr : BOOL ;
    Status_B_Segbert_foliow : BOOL ;
    Status_B_Segbert_deklow : BOOL ;
    Status_B_Segbert_W_wzdl : BOOL ;
    Status_B_Segbert_W_poprz : BOOL ;
    Status_B_Segbert_widoczn : BOOL ;
    res : BOOL ;
    res1 : BOOL ;
    Status_B_Obr_0st_uzbr : BOOL ;
    Status_B_Obr_0st_foliow : BOOL ;
    Status_B_Obr_0st_deklow : BOOL ;
    Status_B_Obr_0st_W_wzdl : BOOL ;
    Status_B_Obr_0st_W_poprz : BOOL ;
    Status_B_Obr_0st_widoczn : BOOL ;
    res2 : BOOL ;
    res3 : BOOL ;
    Status_B_Winda_uzbr : BOOL ;
    Status_B_Winda_foliow : BOOL ;
    Status_B_Winda_deklow : BOOL ;
    Status_B_Winda_W_wzdl : BOOL ;
    Status_B_Winda_W_poprz : BOOL ;
    Status_B_Winda_widoczn : BOOL ;
    res10 : BOOL ;
    res11 : BOOL ;
    Status_B_Wozek_uzbr : BOOL ;
    Status_B_Wozek_foliow : BOOL ;
    Status_B_Wozek_deklow : BOOL ;
    Status_B_Wozek_W_wzdl : BOOL ;
    Status_B_Wozek_W_poprz : BOOL ;
    Status_B_Wozek_widoczn : BOOL ;
    res4 : BOOL ;
    res5 : BOOL ;
    Status_B_Wylot2_uzbr : BOOL ;
    Status_B_Wylot2_foliow : BOOL ;
    Status_B_Wylot2_deklow : BOOL ;
    Status_B_Wylot2_W_wzdl : BOOL ;
    Status_B_Wylot2_W_poprz : BOOL ;
    Status_B_Wylot2_widoczn : BOOL ;
    res6 : BOOL ;
    res7 : BOOL ;
    Status_B_Obr_90st_uzbr : BOOL ;
    Status_B_Obr_90st_foliow : BOOL ;
    Status_B_Obr_90st_deklow : BOOL ;
    Status_B_Obr_90st_W_wzdl : BOOL ;
    Status_B_Obr_90st_W_popr : BOOL ;
    Status_B_Obr_90st_widocz : BOOL ;
    res8 : BOOL ;
    res9 : BOOL ;
    Winda_Dol : BOOL ;
    Winda_Srodek_Dol : BOOL ;
    Winda_Srodek_Gora : BOOL ;
    Winda_Gora : BOOL ;
    Paleta_Winda_Inf_KB2 : DINT ;
    Paleta_Ruch_Pion : INT ;
    Paleta_Ruch_Poziom : INT ;
    Paleta_Winda_Inf_KB2_HMI : DINT ;
    Tablica_IN_INT : ARRAY  [1 .. 13 ] OF INT ;
    Tablica_IN_DWORD : ARRAY  [1 .. 8 ] OF DINT ;
    Aktualna_Data : DATE_AND_TIME ;
   END_STRUCT ;
   HMI_OUT : STRUCT 	//Zmienne wychodzace z HMI Nie nadpisywane w sterowniku od 100 bajta
    Tryb_Uzbrajania_Palety : BOOL ;	//Paleta bedzie uzbrajana dbx100.0
    Tryb_Pracy_Inline : BOOL ;	//Kierunek wylotu palety 1-winda 0-bok dbx100.1
    Ladunek_Na_Intro : BOOL ;	//Reset bledow maszyny
    Reserwa_11 : BOOL ;
    Reserwa_12 : BOOL ;
    Reset_Bledow : BOOL ;	//Reset bledow maszyny
    Reserwa_14 : BOOL ;
    Reserwa_15 : BOOL ;
    Reserwa_16 : BOOL ;
    Reserwa_17 : BOOL ;
    Reserwa_18 : BOOL ;
    Reserwa_19 : BOOL ;
    Reserwa_110 : BOOL ;
    Reserwa_111 : BOOL ;
    Reserwa_112 : BOOL ;
    Reserwa_113 : BOOL ;
    Wybrano_Kier_Spedycje : BOOL ;	//Jedzie na Gender ( dbx2.0)
    Wybrano_Kier_Intro : BOOL ;	//Jedzie na bandy buffory
    Wybrano_Wiaz_Pop : BOOL ;
    Wybrano_Wiaz_Wzdlu : BOOL ;	//Wybrano wiazanie wzdluzne
    Wybrano_Deklowanie : BOOL ;	//wybrano deklowanie
    Wybrano_Foliowanie : BOOL ;
    Kier_Spedycja_Aktywny : BOOL ;
    Kierunek_Intro_Aktywny : BOOL ;
    Wiazanie_Pop_Aktywne : BOOL ;
    Wiazanie_Wzdl_Aktywne : BOOL ;
    Deklowanie_Aktywne : BOOL ;
    Foliowanie_Aktywne : BOOL ;
    reserwa : BOOL ;
    reserwa1 : BOOL ;
    reserwa2 : BOOL ;
    reserwa3 : BOOL ;
    reserwa4 : INT ;	//Wartosc % predkosci z ladunkiem
    Predkosc_Cargo : INT ;	//Wartosc % predkosci z ladunkiem
    Tablica_OUT_INT : ARRAY  [1 .. 21 ] OF INT ;
    Maska_Zadania : INT ;
    Tablica_OUT_DWORD : ARRAY  [1 .. 9 ] OF DWORD ;
    Reserwa_DWORD : DWORD ;
    Aktualna_Data : DATE_AND_TIME ;
   END_STRUCT ;
   HMI_IN_OUT : STRUCT 	//Zmienne nadpisywane w sterowniku i w HMI od 200 bajta
    Reserwa_in_out : BOOL ;
    io_Reserwa : INT ;	//Rodzaj wybranego wlotu
    Predkosc_Obrotnicy : DINT  := L#20;	//dbd4
    Tablica_IN_OUT_INT : ARRAY  [1 .. 22 ] OF INT ;
    Tablica_IN_OUT_DWORD : ARRAY  [1 .. 10 ] OF DWORD ;
    Aktualna_Data : DATE_AND_TIME ;
   END_STRUCT ;
  END_STRUCT ;	
BEGIN
   HMI_IN_OUT.Predkosc_Obrotnicy := L#20;
END_DATA_BLOCK

DATA_BLOCK "DB_HMI_BUF"	// DB 123
AUTHOR : Kng
NAME : HMI_BUFF
VERSION : 0.1
  STRUCT
   HMI_IN : STRUCT 	//Zmienne wchodzace do HMI nie nadpisywane W HMI (100 bajtow)
    Linia_Buffory_Auto : BOOL ;	//Linia buforow jest auto
    Linia_Buffory_Reczny : BOOL ;	//Linia buforow jest w recznym
    Zawsze_True : BOOL ;
    Zawsze_False : BOOL ;
    res255 : BOOL ;
    res54 : BOOL ;
    res11 : BOOL ;
    re32 : BOOL ;
    ret : BOOL ;
    rettt : BOOL ;
    zxc : BOOL ;
    fd : BOOL ;
    zz : BOOL ;
    ddd : BOOL ;
    rrr : BOOL ;
    ttt : BOOL ;
    Linia_Gender_Online : BOOL ;
    Linia_Gender_Offline : BOOL ;
    Linia_Gender_Blad : BOOL ;
    Linia_Blad_Komunikacji : BOOL ;
    Linia_Gender_Auto : BOOL ;
    Linia_Gender_Reczny : BOOL ;
    Linia_Gender_Mark_Bezp : BOOL ;
    Rezerwa_17 : BOOL ;
    Rezerwa_18 : BOOL ;
    Rezerwa_19 : BOOL ;
    Rezerwa_110 : BOOL ;
    Rezerwa_111 : BOOL ;
    Rezerwa_112 : BOOL ;
    Rezerwa_113 : BOOL ;
    Rezerwa_114 : BOOL ;
    Rezerwa_115 : BOOL ;
    Rezerwa_116 : BOOL ;
    I1_Wybor_Kier_Sped : BOOL ;
    I1_Wybor_Kier_Intro : BOOL ;
    I1_Wybor_Wiaz_Pop : BOOL ;
    I1_Wybor_Wiaz_Wzdl : BOOL ;
    I1_Wybor_Deklowanie : BOOL ;
    I1_Wybor_Foliowanie : BOOL ;
    Rezerwa_200 : BOOL ;
    Rezerwa_2001 : BOOL ;
    Rezerwa_2002 : BOOL ;
    Rezerwa_2003 : BOOL ;
    Rezerwa_2004 : BOOL ;
    Rezerwa_2005 : BOOL ;
    Rezerwa_2006 : BOOL ;
    Rezerwa_2007 : BOOL ;
    Rezerwa_2008 : BOOL ;
    rezerwa2009 : BOOL ;
    I2_Wybor_Kier_Sped : BOOL ;
    I2_Wybor_Kier_Intro : BOOL ;
    I2_Wybor_Wiaz_Pop : BOOL ;
    I2_Wybor_Wiaz_Wzdl : BOOL ;
    I2_Wybor_Deklowanie : BOOL ;
    I2_Wybor_Foliowanie : BOOL ;
    Rezerwa_2010 : BOOL ;
    Rezerwa_2011 : BOOL ;
    I3_Wybor_Kier_Sped : BOOL ;
    I3_Wybor_Kier_Intro : BOOL ;
    I3_Wybor_Wiaz_Pop : BOOL ;
    I3_Wybor_Wiaz_Wzdl : BOOL ;
    I3_Wybor_Deklowanie : BOOL ;
    I3_Wybor_Foliowanie : BOOL ;
    Tablica_IN_INT : ARRAY  [1 .. 24 ] OF INT ;
    Tablica_IN_DWORD : ARRAY  [1 .. 9 ] OF DINT ;
    Aktualna_Data : DATE_AND_TIME ;
   END_STRUCT ;
   HMI_OUT : STRUCT 	//Zmienne wychodzace z HMI Nie nadpisywane w sterowniku od 100 bajta
    Zalacz_Buffory_Auto : BOOL ;
    Zalacz_Buffory_Reczny : BOOL ;
    Ladunek_Na_Intro : BOOL ;
    Reserwa_11 : BOOL ;
    Reserwa_12 : BOOL ;
    Reset_Bledow : BOOL ;	//Reset bledow
    Reserwa_14 : BOOL ;
    Reserwa_15 : BOOL ;
    Zalacz_Gender_Online : BOOL ;
    Zalacz_Gender_OFFline : BOOL ;
    Reserwa_18 : BOOL ;
    Reserwa_19 : BOOL ;
    Reserwa_110 : BOOL ;
    Reserwa_111 : BOOL ;
    Reserwa_112 : BOOL ;
    Reserwa_113 : BOOL ;
    I1_Wybrano_Kier_Sped : BOOL ;	//Jedzie na Gender
    I1_Wybrano_Kier_Intro : BOOL ;	//Jedzie na bandy buffory
    I1_Wybrano_Wiaz_Pop : BOOL ;
    I1_Wybrano_Wiaz_Wzdl : BOOL ;	//Wybrano wiazanie wzdluzne
    I1_Wybrano_Dekl : BOOL ;	//wybrano deklowanie
    I1_Wybrano_Foliowanie : BOOL ;
    I1_Kier_Sped_Aktywny : BOOL ;
    I1_Kier_Intro_Aktywny : BOOL ;
    I1_Wiaz_Pop_Aktywne : BOOL ;
    I1_Wiaz_Wzdl_Aktywne : BOOL ;
    I1_Dekl_Aktywne : BOOL ;
    I1_Foliow_Aktywne : BOOL ;
    reserwa : BOOL ;
    reserwa1 : BOOL ;
    reserwa2 : BOOL ;
    VPB_Banda_S_i_2_Tyl : BOOL ;
    VPB_Banda_Shuttle_i_2 : BOOL ;	//Banda reczny Shuttle i 2
    VPB_Banda_2_i_3 : BOOL ;	//banda reczny 2 i 3
    VPB_Banda_3_i_4 : BOOL ;	//banda reczny 3 i 4
    VPB_Banda_4_i_5 : BOOL ;	//banda reczny 4 i 5
    VPB_Banda_5_i_6 : BOOL ;	//banda reczny 5 i 6
    resv_1 : BOOL ;
    resv_11 : BOOL ;
    resv_12 : BOOL ;
    VPB_Banda_12_i_13 : BOOL ;	//Banda reczny 12 i 13
    VPB_Banda_13_i_14 : BOOL ;	//Banda reczny 13 i 14
    VPB_Banda_14_i_15 : BOOL ;	//Banda reczny 14 i 15
    VPB_Banda_15_i_16 : BOOL ;	//Banda reczny 15 i 16
    VPB_Banda_16_i_Shuttle : BOOL ;	//Banda reczny 16 i Shuttle
    VPB_Banda_16_i_S_Tyl : BOOL ;
    Predkosc_Cargo : INT ;	//Wartosc % predkosci z ladunkiem
    rezerwa_6_1 : BOOL ;
    rezerwa_6_2 : BOOL ;
    rezerwa_6_21 : BOOL ;
    rezerwa_6_22 : BOOL ;
    rezerwa_6_23 : BOOL ;
    rezerwa_6_24 : BOOL ;
    rezerwa_6_25 : BOOL ;
    rezerwa_6_26 : BOOL ;
    I2_Wybrano_Kier_Sped : BOOL ;	//Jedzie na Gender
    I2_Wybrano_Kier_Intro : BOOL ;	//Jedzie na bandy buffory
    I2_Wybrano_Wiaz_Pop : BOOL ;
    I2_Wybrano_Wiaz_Wzdl : BOOL ;	//Wybrano wiazanie wzdluzne
    I2_Wybrano_Dekl : BOOL ;	//wybrano deklowanie
    I2_Wybrano_Foliowanie : BOOL ;
    I2_Kier_Sped_Aktywny : BOOL ;
    I2_Kier_Intro_Aktywny : BOOL ;
    I2_Wiaz_Pop_Aktywne : BOOL ;
    I2_Wiaz_Wzdl_Aktywne : BOOL ;
    I2_Dekl_Aktywne : BOOL ;
    I2_Foliow_Aktywne : BOOL ;
    rezerwa_10_4 : BOOL ;
    rezerwa_10_41 : BOOL ;
    rezerwa_10_42 : BOOL ;
    rezerwa_10_43 : BOOL ;
    I3_Wybrano_Kier_Sped : BOOL ;	//Jedzie na Gender
    I3_Wybrano_Kier_Intro : BOOL ;	//Jedzie na bandy buffory
    I3_Wybrano_Wiaz_Pop : BOOL ;
    I3_Wybrano_Wiaz_Wzdl : BOOL ;	//Wybrano wiazanie wzdluzne
    I3_Wybrano_Dekl : BOOL ;	//wybrano deklowanie
    I3_Wybrano_Foliowanie : BOOL ;
    I3_Kier_Sped_Aktywny : BOOL ;
    I3_Kier_Intro_Aktywny : BOOL ;
    I3_Wiaz_Pop_Aktywne : BOOL ;
    I3_Wiaz_Wzdl_Aktywne : BOOL ;
    I3_Dekl_Aktywne : BOOL ;
    I3_Foliow_Aktywne : BOOL ;
    Tablica_OUT_INT : ARRAY  [1 .. 18 ] OF INT ;
    I1_Maska_Zadania : INT ;
    I2_Maska_Zadania : INT ;
    I3_Maska_Zadania : INT ;
    Tablica_OUT_DWORD : ARRAY  [1 .. 8 ] OF DWORD ;
    Reserwa_DWORD : DWORD ;
    Aktualna_Data : DATE_AND_TIME ;
   END_STRUCT ;
   HMI_IN_OUT : STRUCT 	//Zmienne nadpisywane w sterowniku i w HMI od 200 bajta
    Reserwa_in_out : BOOL ;
    io_Tryb_Wlotu : INT ;	//Rodzaj wybranego wlotu
    Tablica_IN_OUT_INT : ARRAY  [1 .. 24 ] OF INT ;
    Tablica_IN_OUT_DWORD : ARRAY  [1 .. 10 ] OF DWORD ;
    Aktualna_Data : DATE_AND_TIME ;
   END_STRUCT ;
  END_STRUCT ;	
BEGIN
END_DATA_BLOCK

DATA_BLOCK "DB_HMI_Wozek"	// DB 128
AUTHOR : Kng
NAME : HMI_WOZ
VERSION : 0.1
  STRUCT
   HMI_IN : STRUCT 	//Zmienne wchodzace do HMI nie nadpisywane W HMI (100 bajtow) PLC-->HMI
    Komunikacja_Wozek_OK : BOOL ;	//### Komunikacja z wozkiem ok
    Wozek_W_Trybie_Auto : BOOL ;	//### Wozek znajduje sie w trybie auto
    Wozek_W_Trybie_Recznym : BOOL ;	//### Wozek znajduje sie w trybie recznym
    Wozek_Petla_0_OK : BOOL ;	//Petla bezpieczenstwa wozka ok
    Wozek_Petla_1_Ok : BOOL ;	//Petla bezpieczenstwa wozka ok
    Wozek_Zasprzeglony : BOOL ;	//### Wozek jest zasprzeglony z banda
    Wozek_Rozprzeglony : BOOL ;	//Wozek jest rozprzeglony z banda
    Wozek_Jest_W_Bledzie : BOOL ;	//### Wozek ma blad
    Pozycja_We_WY_KB1 : BOOL ;
    Pozycja_We_Wy_KB2 : BOOL ;
    Pozycja_We_Wy_Buffory : BOOL ;
    Pozycja_We_Wy_Gender : BOOL ;
    Rezerwa_191 : BOOL ;
    Rezerwa_1101 : BOOL ;
    Wozek_Banda_Lewo : BOOL ;
    Wozek_Banda_Prawo : BOOL ;
    Blokada_I1_Aktywna : BOOL ;	//Blokada Intro wlot I1 aktywna
    Blokada_I2_Aktywna : BOOL ;	//Blokada Intro wlot I2 aktywny
    Blokada_I3_Aktywna : BOOL ;	//Blokada Intro wlot I3 aktywny
    Rezerwa_1161 : BOOL ;
    Rezerwa_112 : BOOL ;
    Rezerwa_113 : BOOL ;
    Rezerwa_114 : BOOL ;
    Rezerwa_115 : BOOL ;
    Wybrana_Strefa_1_Przod : BOOL ;	//Strefa 1 Skaner Przod (<--Shuttle) (dbx3.0)
    Wybrana_Strefa_2_Przod : BOOL ;	//Strefa 2 Skaner Przod (<--Shuttle)
    Wybrana_Strefa_3_Przod : BOOL ;	//Strefa 3 Skaner Przod (<--Shuttle)
    Wybrana_Strefa_4_Przod : BOOL ;	//Strefa 4 Skaner Przod (<--Shuttle)
    Wybrana_Strefa_1_Tyl : BOOL ;	//Strefa 1 Skaner Tyl(<--Shuttle)
    Wybrana_Strefa_2_Tyl : BOOL ;	//Strefa 2 Skaner Tyl (<--Shuttle)
    Wybrana_Strefa_3_Tyl : BOOL ;	//Strefa 3 Skaner Tyl (<--Shuttle)
    Wybrana_Strefa_4_Tyl : BOOL ;	//Strefa 4 Skaner Tyl (<--Shuttle)
    Pozycja_Aktualna : DINT ;	//###
    Rezerwa_222 : BOOL ;
    rezerwa_int : INT ;
    Nr_Bledu_Sew : INT ;	//Blad specyficzny sew do odczytania
    Prad_Aktualny : INT ;	//Prad aktualny SEW
    Predkosc_Aktualna_Wozek : INT ;	//Predkosc akutualna wozka
    Wartosc_Iteracji_Petli : INT ;
    Tablica_IN_INT : ARRAY  [1 .. 18 ] OF INT ;
    Tablica_IN_DWORD : ARRAY  [1 .. 9 ] OF DINT ;
    Aktualna_Data : DATE_AND_TIME ;
   END_STRUCT ;
   HMI_OUT : STRUCT 	//Zmienne wychodzace z HMI Nie nadpisywane w sterowniku (od 100 bajta ) HMI-->PLC
    rezerwaa : BOOL ;
    Przycisk_Wozek_Auto : BOOL ;	//Przycisk wozek auto (dbx100.1)
    Przycisk_Wozek_Reczny : BOOL ;	//Przycisk wozek reczny
    Przycisk_Wozek_Reset : BOOL ;	//Reset bledow wozek
    Przycisk_Wozek_Stop : BOOL ;	//Zatrzymanie zadania wozka
    Reset_Bledow : BOOL ;	//Reset bledow maszyny
    Reserwa_16 : BOOL ;
    Ladunek_Na_Intro : BOOL ;
    Reserwa122 : BOOL ;
    reserwa123 : BOOL ;
    Reserwa_110 : BOOL ;
    Reserwa_111 : BOOL ;
    Reserwa_112 : BOOL ;
    Reserwa_113 : BOOL ;
    reserwa : BOOL ;
    reserwa1 : BOOL ;
    PB_Blokada_Pob_I1 : BOOL ;	//Zablokowaniec pobierania z intro
    PB_Blokada_Pob_I2 : BOOL ;	//Zablokowaniec pobierania z intro
    PB_Blokada_Pob_I3 : BOOL ;	//Zablokowaniec pobierania z intro
    Pozycja_Rezerwa : DINT ;
    Jedz_Na_Pozycje_KB1 : BOOL ;	//###
    Jedz_Na_Pozycje_KB2 : BOOL ;	//###
    Jedz_Na_Pozycje_Gender : BOOL ;	//###
    Jedz_Na_Pozycje_Odbior : BOOL ;	//###
    Jedz_Na_Pozycje_Pob_I1 : BOOL ;	//###
    Jedz_Na_Pozycje_Zadana : BOOL ;	//###
    Jedz_Na_Pozycje_Pob_I2 : BOOL ;
    Jedz_Na_Pozycje_Pob_I3 : BOOL ;
    r12 : BOOL ;
    r13 : BOOL ;
    r14 : BOOL ;
    r15 : BOOL ;
    r16 : BOOL ;
    r17 : BOOL ;
    r18 : BOOL ;
    r19 : BOOL ;
    Pozycja_5_Down : BOOL ;	//(dbx105.0)
    Pozycja_4_Up : BOOL ;
    Pozycja_4_Down : BOOL ;
    Pozycja_3_Up : BOOL ;
    Pozycja_3_Down : BOOL ;
    Pozycja_2_Up : BOOL ;
    Pozycja_2_Down : BOOL ;
    Pozycja_1_Up : BOOL ;
    r20 : BOOL ;
    Wartosc_Stosu_Elem_5 : INT ;
    Wartosc_Stosu_Elem_4 : INT ;
    Wartosc_Stosu_Elem_3 : INT ;
    Wartosc_Stosu_Elem_2 : INT ;
    Wartosc_Stosu_Elem_1 : INT ;
    Wartosc_Akutalnego_Kursu : INT ;
    r21 : BOOL ;
    r211 : BOOL ;
    r212 : BOOL ;
    r213 : BOOL ;
    r214 : BOOL ;
    r215 : BOOL ;
    r216 : BOOL ;
    r217 : BOOL ;
    r218 : BOOL ;
    r219 : BOOL ;
    r2110 : BOOL ;
    r2111 : BOOL ;
    r2112 : BOOL ;
    r2113 : BOOL ;
    r2114 : BOOL ;
    Reset_Para : BOOL ;
    PB_Default_Kier_KB1 : BOOL ;	//przycisk default kierunek rot-kb1
    PB_Move_Default_Kier_KB1 : BOOL ;	//Przycisk przesuwa wartosci z bloku 800 do 801
    PB_Write_Kier_KB1 : BOOL ;	//przycisk zapisania wartosc
    PB_Read_Kier_KB1 : BOOL ;	//przycisk odczytu wartosci
    PB_Move_Read_Kier_KB1 : BOOL ;	//przesuwa wartosc z db802 do db801
    PB_Save_Default_Kier_KB1 : BOOL ;	//zapisz do defaultowych
    Aktywny_Ekran_Kier_KB1 : BOOL ;
    res_kier_Kb11 : BOOL ;
    PB_Default_Kier_Rot : BOOL ;	//przycisk default kierunek
    PB_Move_Default_Kier_Rot : BOOL ;	//Przycisk przesuwa wartosci z bloku 800 do 801
    PB_Write_Kier_Rot : BOOL ;	//przycisk zapisania wartosc
    PB_Read_Kier_Rot : BOOL ;	//przycisk odczytu wartosci
    PB_Move_Read_Kier_Rot : BOOL ;	//przesuwa wartosc z db802 do db801
    PB_Save_Default_Kier_Rot : BOOL ;	//zapisuje do defaulta
    Aktywny_Ekran_Kier_Rot : BOOL ;
    res_kier_Kb13 : BOOL ;
    PB_Default_Para : BOOL ;	//przycisk default kierunek
    PB_Move_Default_Para : BOOL ;	//Przycisk przesuwa wartosci z bloku 800 do 801
    PB_Write_Para : BOOL ;	//przycisk zapisania wartosc
    PB_Read_Para : BOOL ;	//przycisk odczytu wartosci
    PB_Move_Read_Para : BOOL ;	//przesuwa wartosc z db802 do db801
    PB_Save_Default_Para : BOOL ;	//zapisuje parametry do defaultu
    Aktywny_Ekran_Kier_Para : BOOL ;
    res_kier_Kb15 : BOOL ;
    reserwa_int_1 : INT ;	//Wartosc iteracji wymienianych danych
    PB_Default_Odb : BOOL ;	//przycisk default kierunek
    PB_Move_Default_Odb : BOOL ;	//Przycisk przesuwa wartosci z bloku 800 do 801
    PB_Write_Odb : BOOL ;	//przycisk zapisania wartosc
    PB_Read_Odb : BOOL ;	//przycisk odczytu wartosci
    PB_Move_Read_Odb : BOOL ;	//przesuwa wartosc z db802 do db801
    PB_Save_Default_Odb : BOOL ;	//zapisuje parametry do defaultu
    Aktywny_Ekran_Odb : BOOL ;
    res_kier_Kb151 : BOOL ;
    Tablica_OUT_INT : ARRAY  [1 .. 12 ] OF INT ;
    Maska_Zadania : INT ;
    Tablica_OUT_DWORD : ARRAY  [1 .. 7 ] OF DWORD ;
    Reserwa_DWORD : DWORD ;
    Aktualna_Data : DATE_AND_TIME ;
   END_STRUCT ;
   HMI_IN_OUT : STRUCT 	//Zmienne nadpisywane w sterowniku i w HMI od 200 bajta
    Reserwa_in_out : BOOL ;
    rez_int : INT ;
    Pozycja_Zadana : DINT ;	//### Pozycja zadawana z HMI lub zadawana z PLC (dbd204)
    Wartosc_Buforu_Wozek : DINT ;
    Wartosc_Wozek_HMI : DINT ;	//Wartosc wozek dla HMI
    Wartosc_Wozek_HMI_HMI : DINT ;	//Wartosc wozek dla HMI
    Tablica_IN_OUT_INT : ARRAY  [1 .. 20 ] OF INT ;
    Tablica_IN_OUT_DWORD : ARRAY  [1 .. 8 ] OF DWORD ;
    Aktualna_Data : DATE_AND_TIME ;
   END_STRUCT ;
  END_STRUCT ;	
BEGIN
END_DATA_BLOCK

DATA_BLOCK "COM_SHUTTLE"	// DB 200
VERSION : 0.1
  STRUCT
   IN : STRUCT
    Bit_Kom_Shuttle : BOOL ;	//Bit toggle komunikacji z wozkiem (<--)Shuttle
    Petla_Bezp_0_OK : BOOL ;	//Petla bezpieczenstwa 0 OK (<--Shuttle )
    Petla_Bezp_1_OK : BOOL ;	//Petla bezpieczenstwa 1 OK ( <--Shuttle)
    Wozek_Auto_Info : BOOL ;	//Wozek w Auto - 1 lub Reczny - 2
    Blad_Wozka : BOOL ;	//Wozek jest w bledzie
    Falownik_Band_Gotowy : BOOL ;	//Falownik band gotowy
    PB_Reset : BOOL ;	//Przycisk reset wozek
    Res_0_7 : BOOL ;
    Bit_Com_od_Shuttle : BOOL ;
    Potw_Nowej_Pozycji : BOOL ;	//Bit potwierdzenia przyjecia nowej pozycji (<-- Shuttle )
    Shuttle_Na_Pozycji : BOOL ;	//Wozek na pozycji (<--Shuttle )
    Shuttle_Stoi : BOOL ;	//Wozek na pozycji (Shuttle <--)
    Potw_Zasprz : BOOL ;	//Potwierdzenie zasprzeglenia (<--)Shuttle
    Potw_Rozprz : BOOL ;	//Potwierdzenie Rozprzeglenia (<--Shuttle )
    Foto_Przod : BOOL ;	//Fotokomorka wozek przod (<--Shuttle )
    Foto_Wozek_Tyl : BOOL ;	//Fotokomorka wozek tyl (<--Shuttle)
    Res_2_0 : BOOL ;
    Res_2_1 : BOOL ;
    Res_2_2 : BOOL ;
    Res_2_3 : BOOL ;
    Res_2_4 : BOOL ;
    Res_2_5 : BOOL ;
    Res_2_6 : BOOL ;
    Res_2_7 : BOOL ;
    Wybrana_Strefa_1_Przod : BOOL ;	//Strefa 1 Skaner Przod (<--Shuttle)
    Wybrana_Strefa_2_Przod : BOOL ;	//Strefa 2 Skaner Przod (<--Shuttle)
    Wybrana_Strefa_3_Przod : BOOL ;	//Strefa 3 Skaner Przod (<--Shuttle)
    Wybrana_Strefa_4_Przod : BOOL ;	//Strefa 4 Skaner Przod (<--Shuttle)
    Wybrana_Strefa_1_Tyl : BOOL ;	//Strefa 1 Skaner Tyl(<--Shuttle)
    Wybrana_Strefa_2_Tyl : BOOL ;	//Strefa 2 Skaner Tyl (<--Shuttle)
    Wybrana_Strefa_3_Tyl : BOOL ;	//Strefa 3 Skaner Tyl (<--Shuttle)
    Wybrana_Strefa_4_Tyl : BOOL ;	//Strefa 4 Skaner Tyl (<--Shuttle)
    Poz_Akt_Wozka : DINT ;	//Pozycja aktualna wozka
   END_STRUCT ;
   OUT : STRUCT
    Bit_Kom_Odbieranie : BOOL ;	//Bit komunikacji do Shuttle(-->Shuttle)
    Bit_Bezpieczenstwa_0 : BOOL ;	//Bit bezpieczenstwa 0 (-->Shuttle)
    Reset_Wozka : BOOL ;	//Bit Resetu Shuttle ( -->Shuttle)
    Wozek_Auto : BOOL ;	//Bit ustawienia wozka Auto
    Wozek_Reczny : BOOL ;	//Bit ustwienia Reczny
    Partner_Reczny : BOOL ;	//Partner wozka reczny i wozek przejmuje to
    Reset_Zadania : BOOL ;	//Reset Zadania Wozka
    Res_0_7 : BOOL ;
    Bit_Com_do_Shuttle : BOOL ;
    op_Bit_Nowej_Pozycji : BOOL ;	//Bit zadania nowej pozycji (-->Shuttle)
    op_Potw_Pozycji : BOOL ;	//Bit potwierdzenia pozycji (-->Shuttle)
    Rez_1_3 : BOOL ;
    op_Zasprz_Wozka : BOOL ;	//Rozkaz Zasprzeglenie Wozka (-->Shuttle)
    op_Rozprz_Wozka : BOOL ;	//Rozkaz Rozprzeglenie Wozka (--> Shuttle)
    op_Silnik_Banda_Lewo : BOOL ;	//Jazda silnika w lewo (-->Shuttle)
    op_Silnik_Banda_Prawo : BOOL ;	//Jazda silnika w prawo (-->Shuttle)
    Res_2_0 : BOOL ;
    Res_2_1 : BOOL ;
    Res_2_2 : BOOL ;
    Res_2_3 : BOOL ;
    Res_2_4 : BOOL ;
    Res_2_5 : BOOL ;
    Res_2_6 : BOOL ;
    Res_2_7 : BOOL ;
    Pozycja_KB1 : BOOL ;	//Blokada dalekiej jazdy w prawo
    Pozycja_KB2 : BOOL ;	//Blokada dalekiej jazdy w prawo
    Pozycja_Gender : BOOL ;	//Blokada dalekiej jazdy w lewo
    Pozycja_Intro_Pob_I1 : BOOL ;	//Blokada dalekiej jazdy w lewo
    Pozycja_Intro_Odb : BOOL ;	//Blokada dalekiej jazdy w lewo
    Pozycja_Intro_Pob_I2 : BOOL ;	//Blokada dalekiej jazdy w prawo
    Pozycja_Intro_Pob_I3 : BOOL ;	//Blokada dalekiej jazdy w prawo
    Res_3_7 : BOOL ;
    Pozycja_Zadana : DINT ;	//Pozycja zadana w mm (--> Shuttle)
   END_STRUCT ;
   SOME_IN : STRUCT
    tab_32 : ARRAY  [1 .. 32 ] OF BYTE ;
   END_STRUCT ;
   SOME_OUT : STRUCT
    tab_32 : ARRAY  [1 .. 32 ] OF BYTE ;
   END_STRUCT ;
  END_STRUCT ;	
BEGIN
END_DATA_BLOCK

DATA_BLOCK "LLOUT"	// DB 201
VERSION : 0.1
  STRUCT
   OUT : STRUCT 	//Dane wejsciowe z Odbierania
    Zadanie_Transmisji : BOOL ;
    Zadanie_Danych : BOOL ;
    Toggle : BOOL ;	//bit- in/out
    Rezerwa_0_3 : BOOL ;
    Rezerwa_0_4 : BOOL ;
    Funcja_Receive : BOOL ;
    Funkcja_Share : BOOL ;
    Rezerwa_0_7 : BOOL ;
    Rezerwa_Bajt_1 : BYTE ;
    Nr_Bloku : INT  := 701;	//Nr bloku gdzie dane (read/send)
    Nr_Rekordu : INT ;	//Nr rekordu wysylanego (read/send)
    Kanal_Nadawania : INT ;	//Kanal Nadawania (send)
    Rezerwa_Bajtow : ARRAY  [1 .. 8 ] OF BYTE ;
    Predkosc_Cargo : INT  := 100;	//Predkosc Cargo w procentach
    Reserwa_Dalej : ARRAY  [1 .. 14 ] OF BYTE ;
   END_STRUCT ;
  END_STRUCT ;	
BEGIN
   OUT.Nr_Bloku := 701;
END_DATA_BLOCK

DATA_BLOCK "LLIN"	// DB 202
VERSION : 0.1
  STRUCT
   IN : STRUCT 	//Dane wejsciowe z Odbierania
    Transmisja_Ustanowiona : BOOL ;
    Blok_Zarezerwowany : BOOL ;
    Toggle : BOOL ;	//bit- in/out
    Przesylanie_Danych : BOOL ;
    Koniec_Nadawania : BOOL ;
    Receive_Wybrane : BOOL ;
    Share_Wybrane : BOOL ;
    Rezerwa_0_7 : BOOL ;
    Rezerwa_Bajt_1 : BYTE ;
    Nr_Rekordu : INT  := 701;
    Licznik_Rekordow : INT ;	//Potwierdzenie Rekordu (Share/receive)
    Kanal_Pobierania : INT ;	//Pobieranie danych (Share)
    Rezerwa_Bajtow : ARRAY  [1 .. 8 ] OF BYTE ;
    Bledy_Wozka : ARRAY  [1 .. 16 ] OF
    BYTE ;
   END_STRUCT ;
  END_STRUCT ;	
BEGIN
   IN.Nr_Rekordu := 701;
END_DATA_BLOCK

DATA_BLOCK "COM_GENDER"	// DB 205
VERSION : 0.1
  STRUCT
   IN : STRUCT 	//Temporary placeholder variable
    Bit_Com_Odbieranie : BOOL ;
    Auto_Reczny_Gender : BOOL ;	//1-auto , 0- reczny
    Marka_Bezp_Gender : BOOL ;
    Linia_Gender_Online : BOOL ;	//Linia Gender odbiera palety z shuttle
    Blad_Lini_Gender : BOOL ;	//Linia Gender jest w bledzie
    Res_0_5 : BOOL ;
    PB_Auto : BOOL ;
    PB_Reczny : BOOL ;
    PB_Banda_Wozek_Tyl : BOOL ;
    PB_Banda_Wozek_Przod : BOOL ;
    Banda_1_Gen_Zez_Do_Pop : BOOL ;	//banda gender zezwolenie do porzedniej
    Banda_1_Gen_Pal_Dost : BOOL ;	//Paleta dostarczona
    Banda_1_Gen_Zez_R_Do_Pop : BOOL ;	//zezwolenie reczny do poprzedniej
    Res_1_5 : BOOL ;
    Res_1_6 : BOOL ;
    Res_1_7 : BOOL ;
    Bindownica_Agregat_Auto : BOOL ;
    Res_2_1 : BOOL ;
    Res_2_2 : BOOL ;
    Res_2_3 : BOOL ;
    Res_2_4 : BOOL ;
    Res_2_5 : BOOL ;
    Res_2_6 : BOOL ;
    Res_2_7 : BOOL ;
    Res_3_0 : BOOL ;
    Res_3_1 : BOOL ;
    Res_3_2 : BOOL ;
    Res_3_3 : BOOL ;
    Res_3_4 : BOOL ;
    Res_3_5 : BOOL ;
    Res_3_6 : BOOL ;
    Res_3_7 : BOOL ;
    Zmienna_DINT : DINT ;
   END_STRUCT ;
   OUT : STRUCT 	//Temporary placeholder variable
    Bit_Com_Odbieranie : BOOL ;
    Auto_Reczny_Shuttle : BOOL ;	//1-auto , 0- reczny
    Marka_Bezp_Shuttle : BOOL ;
    Wymuszenie_Online : BOOL ;	//Wymuszenie Lini gender online
    Wymuszenie_Offline : BOOL ;	//Wymuszenie Lini gender offline (wykorzystanie wozka widlowego)
    Wozek_Na_Pozycji_Gender : BOOL ;
    Wozek_Zasprzeglony : BOOL ;
    Res_0_7 : BOOL ;
    Wozek_Zab_do_Nast : BOOL ;	//Wozek zabierz do nastepnej
    Wozek_Zez_R_do_Nast : BOOL ;	//Wozek zezwolenie reczny do nastepnej
    Foto_Wozek_Przod : BOOL ;	//Foto Wozek Przod
    Foto_Wozek_Tyl : BOOL ;	//Foto Wozek Tyl
    Motor_Wozek_Tyl : BOOL ;	//Motor wozek tyl
    Motor_Wozek_Przod : BOOL ;	//Motor wozek przod
    Res_1_6 : BOOL ;
    Res_1_7 : BOOL ;
    Res_2_0 : BOOL ;
    Res_2_1 : BOOL ;
    Res_2_2 : BOOL ;
    Res_2_3 : BOOL ;
    Res_2_4 : BOOL ;
    Res_2_5 : BOOL ;
    Res_2_6 : BOOL ;
    Res_2_7 : BOOL ;
    Res_3_0 : BOOL ;
    Res_3_1 : BOOL ;
    Res_3_2 : BOOL ;
    Res_3_3 : BOOL ;
    Res_3_4 : BOOL ;
    Res_3_5 : BOOL ;
    Res_3_6 : BOOL ;
    Res_3_7 : BOOL ;
    Zmienna_DINT : DINT ;
   END_STRUCT ;
  END_STRUCT ;	
BEGIN
END_DATA_BLOCK

DATA_BLOCK "Stale_Maszynowe"	// DB 300
VERSION : 0.1
  STRUCT
   Pozycja_Skrajna_Dol : DINT  := L#280;
   Pozycja_KB1 : DINT  := L#400;	//Temporary placeholder variable
   Pozycja_KB2 : DINT  := L#15905;
   Pozycja_Gender : DINT  := L#24780;
   Pozycja_odbieranie : DINT  := L#33000;
   Pozycja_Pob_I1 : DINT  := L#34180;
   Pozycja_Skrajna_Gora : DINT  := L#34210;
   Reserwa : DINT ;
   War_W_Kolejce_KB1 : DINT  := L#200;
   War_W_Kolejce_KB2 : DINT  := L#200;
   War_W_Kolejce_I1 : DINT  := L#100;
   War_W_Kolejce_I2 : DINT  := L#100;
   War_W_Kolejce_I3 : DINT  := L#100;
   Pozycja_Pob_I2 : DINT  := L#32944;
   Pozycja_Pob_I3 : DINT  := L#34111;
   Reserwa_21 : DINT ;
   Reserwa_22 : DINT ;
   Reserwa_24 : DINT ;
   res : DINT ;
   res1 : DINT ;
   res2 : DINT ;
   res3 : DINT ;
   res4 : DINT ;
   res5 : DINT ;
   res6 : DINT ;
   res7 : DINT ;
   res8 : DINT ;
   res81 : DINT ;
   res82 : DINT ;
   res83 : DINT ;
   res84 : DINT ;
   res85 : DINT ;
   res86 : DINT ;
   res87 : DINT ;
   res88 : DINT ;
   res89 : DINT ;
   res810 : DINT ;
   res811 : DINT ;
   res812 : DINT ;
   res813 : DINT ;
   res814 : DINT ;
   res815 : DINT ;
   res816 : DINT ;
   res817 : DINT ;
   res818 : DINT ;
   res819 : DINT ;
   res820 : DINT ;
   res821 : DINT ;
   res822 : DINT ;
   res823 : DINT ;
  END_STRUCT ;	
BEGIN
   Pozycja_Skrajna_Dol := L#280;
   Pozycja_KB1 := L#400;
   Pozycja_KB2 := L#15905;
   Pozycja_Gender := L#24780;
   Pozycja_odbieranie := L#33000;
   Pozycja_Pob_I1 := L#34180;
   Pozycja_Skrajna_Gora := L#34210;
   War_W_Kolejce_KB1 := L#200;
   War_W_Kolejce_KB2 := L#200;
   War_W_Kolejce_I1 := L#100;
   War_W_Kolejce_I2 := L#100;
   War_W_Kolejce_I3 := L#100;
   Pozycja_Pob_I2 := L#32944;
   Pozycja_Pob_I3 := L#34111;
END_DATA_BLOCK

DATA_BLOCK "DB_Trace"	// DB 402
VERSION : 0.1
  STRUCT
   Wpis : STRUCT
    _0_dbb0_Kod_Kier : BYTE ;
    _0_dbb1_Kod_Maszyna : BYTE ;
    _0_dbw2_War_Wagowa : INT ;
    _1_dbb4_Kod_Kier : BYTE ;
    _1_dbb5_Kod_Maszyna : BYTE ;
    _1_dbw6_War_Wagowa : INT ;
    _2_dbb8_Kod_Kier : BYTE ;
    _2_dbb9_Kod_Maszyna : BYTE ;
    _2_dbw10_War_Wagowa : INT ;
    _3_dbb12_Kod_Kier : BYTE ;
    _3_dbb13_Kod_Maszyna : BYTE ;
    _3_dbw14_War_Wagowa : INT ;
    _4_dbb16_Kod_Kier : BYTE ;
    _4_dbb17_Kod_Maszyna : BYTE ;
    _4_dbw18_War_Wagowa : INT ;
    _5_dbb20_Wsad_Kod_Kier : BYTE ;
    _5_dbb21_Wsad_Kod_Masz : BYTE ;
    _5_dbw22_Wsad_Waga : INT ;
    Kod_Spr_KB1 : BYTE ;
    Kod_Spr_KB2 : BYTE ;
    Kod_Spr_Intro : BYTE ;
    Kod_Spr_Reserwa : BYTE ;
   END_STRUCT ;
  END_STRUCT ;	
BEGIN
END_DATA_BLOCK

DATA_BLOCK "Key_DB"	// DB 409
VERSION : 0.1
  STRUCT
   Wpis : STRUCT
    _0_dbb0_Kod_Kier : BYTE ;
    _0_dbb1_Kod_Maszyna : BYTE ;
    _0_dbw2_War_Wagowa : INT ;
    _1_dbb4_Kod_Kier : BYTE ;
    _1_dbb5_Kod_Maszyna : BYTE ;
    _1_dbw6_War_Wagowa : INT ;
    _2_dbb8_Kod_Kier : BYTE ;
    _2_dbb9_Kod_Maszyna : BYTE ;
    _2_dbw10_War_Wagowa : INT ;
    _3_dbb12_Kod_Kier : BYTE ;
    _3_dbb13_Kod_Maszyna : BYTE ;
    _3_dbw14_War_Wagowa : INT ;
    _4_dbb16_Kod_Kier : BYTE ;
    _4_dbb17_Kod_Maszyna : BYTE ;
    _4_dbw18_War_Wagowa : INT ;
    _5_dbb20_Kod_Kier : BYTE ;
    _5_dbb21_Kod_Masz : BYTE ;
    _5_dbw22_War_Wagowa : INT ;
    _6_dbb24_Kod_Kier : BYTE ;
    _6_dbb25_Kod_Masz : BYTE ;
    _6_dbw26_War_Wagowa : INT ;
    Kod_Spr_KB1 : BYTE ;
    Kod_Spr_KB2 : BYTE ;
    Kod_Spr_I1 : BYTE ;
    Kod_Spr_I2 : BYTE ;
    Kod_Spr_I3 : BYTE ;
    Kod_Spr_Rezerwa : BYTE ;
   END_STRUCT ;
  END_STRUCT ;	
BEGIN
END_DATA_BLOCK

DATA_BLOCK "Blok_Default"	// DB 800
VERSION : 0.1
  STRUCT
   DB_VAR : ARRAY  [1 .. 300 ] OF //Temporary placeholder variable
   INT  := 0;
  END_STRUCT ;	
BEGIN
END_DATA_BLOCK

DATA_BLOCK "Blok_Write"	// DB 801
VERSION : 0.1
  STRUCT
   DB_VAR : ARRAY  [1 .. 300 ] OF //Temporary placeholder variable
   INT  := 0;
  END_STRUCT ;	
BEGIN
END_DATA_BLOCK

DATA_BLOCK "Blok_Read"	// DB 802
VERSION : 0.1
  STRUCT
   DB_VAR : ARRAY  [1 .. 300 ] OF //Temporary placeholder variable
   INT  := 0;
  END_STRUCT ;	
BEGIN
END_DATA_BLOCK

DATA_BLOCK "Def_Blok_Para_Wozek"	// DB 811
VERSION : 0.1
  STRUCT
   Predkosc_Ostrzegawcza : DINT  := L#50;	//Zmiana predkosci procentowa w strefie ostrzegawczej [50]
   Predkosc_Maksymalna : DINT  := L#300;	//Predkosc maksymalna wozka
   Rampa_Startu_Wozka : DINT  := L#2000;	//Rampa startu wozka [ms]
   Rampa_Stopu_Wozka : DINT  := L#2000;	//Rampa stopu wozka [ms]
   Predkosc_Na_Pelno : DINT  := L#100;	//Predkosc w % wozka pelnego
   DB_VAR3 : DINT  := L#2;	//Temporary placeholder variable
   DB_VAR4 : DINT ;	//Temporary placeholder variable
   DB_VAR5 : DINT ;	//Temporary placeholder variable
   DB_VAR6 : DINT ;	//Temporary placeholder variable
   DB_VAR7 : DINT ;	//Temporary placeholder variable
   DB_VAR8 : DINT ;	//Temporary placeholder variable
   DB_VAR9 : DINT ;	//Temporary placeholder variable
   DB_VAR10 : DINT ;	//Temporary placeholder variable
   DB_VAR11 : DINT ;	//Temporary placeholder variable
   DB_VAR12 : DINT ;	//Temporary placeholder variable
   DB_VAR13 : DINT ;	//Temporary placeholder variable
   DB_VAR14 : DINT ;	//Temporary placeholder variable
   DB_VAR15 : DINT ;	//Temporary placeholder variable
   DB_VAR16 : DINT ;	//Temporary placeholder variable
   DB_VAR17 : DINT ;	//Temporary placeholder variable
   DB_VAR18 : DINT ;	//Temporary placeholder variable
   DB_VAR19 : DINT ;	//Temporary placeholder variable
   DB_VAR191 : DINT ;	//Temporary placeholder variable
   DB_VAR192 : DINT ;	//Temporary placeholder variable
   DB_VAR193 : DINT ;	//Temporary placeholder variable
   DB_VAR194 : DINT ;	//Temporary placeholder variable
   DB_VAR195 : DINT ;	//Temporary placeholder variable
   DB_VAR1951 : DINT ;	//Temporary placeholder variable
   DB_VAR19511 : DINT ;	//Temporary placeholder variable
   DB_VAR19512 : DINT ;	//Temporary placeholder variable
   DB_VAR19513 : DINT ;	//Temporary placeholder variable
   DB_VAR19514 : DINT ;	//Temporary placeholder variable
   DB_VAR19515 : DINT ;	//Temporary placeholder variable
   DB_VAR19516 : DINT ;	//Temporary placeholder variable
   DB_VAR19517 : DINT ;	//Temporary placeholder variable
   DB_VAR19518 : DINT ;	//Temporary placeholder variable
   DB_VAR19519 : DINT ;	//Temporary placeholder variable
   DB_VAR195110 : DINT ;	//Temporary placeholder variable
   DB_VAR195111 : DINT ;	//Temporary placeholder variable
   DB_VAR195112 : DINT ;	//Temporary placeholder variable
   DB_VAR195113 : DINT ;	//Temporary placeholder variable
   DB_VAR195114 : DINT ;	//Temporary placeholder variable
   DB_VAR195115 : DINT ;	//Temporary placeholder variable
   DB_VAR195116 : DINT ;	//Temporary placeholder variable
   DB_VAR195117 : DINT ;	//Temporary placeholder variable
   DB_VAR195118 : DINT ;	//Temporary placeholder variable
   DB_VAR195119 : DINT ;	//Temporary placeholder variable
   DB_VAR195120 : DINT ;	//Temporary placeholder variable
   DB_VAR195121 : DINT ;	//Temporary placeholder variable
   DB_VAR195122 : DINT ;	//Temporary placeholder variable
  END_STRUCT ;	
BEGIN
   Predkosc_Ostrzegawcza := L#50;
   Predkosc_Maksymalna := L#300;
   Rampa_Startu_Wozka := L#2000;
   Rampa_Stopu_Wozka := L#2000;
   Predkosc_Na_Pelno := L#100;
   DB_VAR3 := L#2;
END_DATA_BLOCK

DATA_BLOCK "Def_Blok_Kier_KB1"	// DB 820
VERSION : 0.1
  STRUCT
   Wartosc_Poz_Kier_KB1 : STRUCT 	//Wartosc pozycji
    Poz_0 : DINT  := L#37000;
    Poz_1 : DINT  := L#33000;
    Poz_2 : DINT  := L#17000;
    Poz_3 : DINT  := L#12000;
    Poz_4 : DINT  := L#9000;
    Poz_5 : DINT  := L#5000;
    Poz_6 : DINT ;
    Poz_7 : DINT ;
    Poz_8 : DINT ;
    Poz_9 : DINT ;
    Poz_10 : DINT ;
    Poz_11 : DINT ;
    Poz_12 : DINT ;
    poz_13 : DINT ;
    Poz_14 : DINT ;
    Poz_15 : DINT ;
    Poz_16 : DINT ;
    Poz_17 : DINT ;
    Poz_18 : DINT ;
    Poz_19 : DINT ;
    Poz_20 : DINT ;
    Poz_21 : DINT ;
    Poz_22 : DINT ;
    poz_23 : DINT ;
    Poz_24 : DINT ;
   END_STRUCT ;
   Wartosc_Strefy : STRUCT 	//Wartosc Strefy
    Strefa_0 : DINT  := L#4;
    Strefa_1 : DINT  := L#4;
    Strefa_2 : DINT  := L#4;
    Strefa_3 : DINT  := L#4;
    Strefa_4 : DINT  := L#4;
    Strefa_5 : DINT  := L#4;
    Strefa_6 : DINT  := L#4;
    Strefa_7 : DINT  := L#4;
    Strefa_8 : DINT  := L#4;
    Strefa_9 : DINT  := L#4;
    Strefa_10 : DINT  := L#4;
    Strefa_11 : DINT  := L#4;
    Strefa_12 : DINT  := L#4;
    Strefa_13 : DINT  := L#4;
    Strefa_14 : DINT  := L#4;
    Strefa_15 : DINT  := L#4;
    Strefa_16 : DINT  := L#4;
    Strefa_17 : DINT  := L#4;
    Strefa_18 : DINT  := L#4;
    Strefa_19 : DINT  := L#4;
    Strefa_20 : DINT  := L#4;
    Strefa_21 : DINT  := L#4;
    Strefa_22 : DINT  := L#4;
    Strefa_23 : DINT  := L#4;
    Strefa_24 : DINT  := L#4;
   END_STRUCT ;
   Wartosc_Predkosci : STRUCT 	//Wartosc Predkosci w procentach
    Predkosc_0 : DINT  := L#100;
    Predkosc_1 : DINT  := L#100;
    Predkosc_2 : DINT  := L#100;
    Predkosc_3 : DINT  := L#100;
    Predkosc_4 : DINT  := L#100;
    Predkosc_5 : DINT  := L#100;
    Predkosc_6 : DINT  := L#100;
    Predkosc_7 : DINT  := L#100;
    Predkosc_8 : DINT  := L#100;
    Predkosc_9 : DINT  := L#100;
    Predkosc_10 : DINT  := L#100;
    Predkosc_11 : DINT  := L#100;
    Predkosc_12 : DINT  := L#100;
    Predkosc_13 : DINT  := L#100;
    Predkosc_14 : DINT  := L#100;
    Predkosc_15 : DINT  := L#100;
    Predkosc_16 : DINT  := L#100;
    Predkosc_17 : DINT  := L#100;
    Predkosc_18 : DINT  := L#100;
    Predkosc_19 : DINT  := L#100;
    Predkosc_20 : DINT  := L#100;
    Predkosc_21 : DINT  := L#100;
    Predkosc_22 : DINT  := L#100;
    Predkosc_23 : DINT  := L#100;
    Predkosc_24 : DINT  := L#100;
   END_STRUCT ;
  END_STRUCT ;	
BEGIN
   Wartosc_Poz_Kier_KB1.Poz_0 := L#37000;
   Wartosc_Poz_Kier_KB1.Poz_1 := L#33000;
   Wartosc_Poz_Kier_KB1.Poz_2 := L#17000;
   Wartosc_Poz_Kier_KB1.Poz_3 := L#12000;
   Wartosc_Poz_Kier_KB1.Poz_4 := L#9000;
   Wartosc_Poz_Kier_KB1.Poz_5 := L#5000;
   Wartosc_Strefy.Strefa_0 := L#4;
   Wartosc_Strefy.Strefa_1 := L#4;
   Wartosc_Strefy.Strefa_2 := L#3;
   Wartosc_Strefy.Strefa_3 := L#4;
   Wartosc_Strefy.Strefa_4 := L#4;
   Wartosc_Strefy.Strefa_5 := L#4;
   Wartosc_Strefy.Strefa_6 := L#4;
   Wartosc_Strefy.Strefa_7 := L#4;
   Wartosc_Strefy.Strefa_8 := L#4;
   Wartosc_Strefy.Strefa_9 := L#4;
   Wartosc_Strefy.Strefa_10 := L#4;
   Wartosc_Strefy.Strefa_11 := L#4;
   Wartosc_Strefy.Strefa_12 := L#4;
   Wartosc_Strefy.Strefa_13 := L#4;
   Wartosc_Strefy.Strefa_14 := L#4;
   Wartosc_Strefy.Strefa_15 := L#4;
   Wartosc_Strefy.Strefa_16 := L#4;
   Wartosc_Strefy.Strefa_17 := L#4;
   Wartosc_Strefy.Strefa_18 := L#4;
   Wartosc_Strefy.Strefa_19 := L#4;
   Wartosc_Strefy.Strefa_20 := L#4;
   Wartosc_Strefy.Strefa_21 := L#4;
   Wartosc_Strefy.Strefa_22 := L#4;
   Wartosc_Strefy.Strefa_23 := L#4;
   Wartosc_Strefy.Strefa_24 := L#4;
   Wartosc_Predkosci.Predkosc_0 := L#100;
   Wartosc_Predkosci.Predkosc_1 := L#100;
   Wartosc_Predkosci.Predkosc_2 := L#100;
   Wartosc_Predkosci.Predkosc_3 := L#100;
   Wartosc_Predkosci.Predkosc_4 := L#100;
   Wartosc_Predkosci.Predkosc_5 := L#100;
   Wartosc_Predkosci.Predkosc_6 := L#100;
   Wartosc_Predkosci.Predkosc_7 := L#100;
   Wartosc_Predkosci.Predkosc_8 := L#100;
   Wartosc_Predkosci.Predkosc_9 := L#100;
   Wartosc_Predkosci.Predkosc_10 := L#100;
   Wartosc_Predkosci.Predkosc_11 := L#100;
   Wartosc_Predkosci.Predkosc_12 := L#100;
   Wartosc_Predkosci.Predkosc_13 := L#100;
   Wartosc_Predkosci.Predkosc_14 := L#100;
   Wartosc_Predkosci.Predkosc_15 := L#100;
   Wartosc_Predkosci.Predkosc_16 := L#100;
   Wartosc_Predkosci.Predkosc_17 := L#100;
   Wartosc_Predkosci.Predkosc_18 := L#100;
   Wartosc_Predkosci.Predkosc_19 := L#100;
   Wartosc_Predkosci.Predkosc_20 := L#100;
   Wartosc_Predkosci.Predkosc_21 := L#100;
   Wartosc_Predkosci.Predkosc_22 := L#100;
   Wartosc_Predkosci.Predkosc_23 := L#100;
   Wartosc_Predkosci.Predkosc_24 := L#100;
END_DATA_BLOCK

DATA_BLOCK "Def_Blok_Kier_Rot"	// DB 821
VERSION : 0.1
  STRUCT
   Wartosc_Pozycji : STRUCT 	//Wartosc pozycji
    Poz_0 : DINT ;
    Poz_1 : DINT  := L#1000;
    Poz_2 : DINT  := L#2000;
    Poz_3 : DINT  := L#5000;
    Poz_4 : DINT  := L#20000;
    Poz_5 : DINT  := L#40000;
    Poz_6 : DINT ;
    Poz_7 : DINT ;
    Poz_8 : DINT ;
    Poz_9 : DINT ;
    Poz_10 : DINT ;
    Poz_11 : DINT ;
    Poz_12 : DINT ;
    poz_13 : DINT ;
    Poz_14 : DINT ;
    Poz_15 : DINT ;
    Poz_16 : DINT ;
    Poz_17 : DINT ;
    Poz_18 : DINT ;
    Poz_19 : DINT ;
    Poz_20 : DINT ;
    Poz_21 : DINT ;
    Poz_22 : DINT ;
    poz_23 : DINT ;
    Poz_24 : DINT ;
   END_STRUCT ;
   Wartosc_Strefy : STRUCT 	//Wartosc Strefy
    Strefa_0 : DINT  := L#4;
    Strefa_1 : DINT  := L#4;
    Strefa_2 : DINT  := L#4;
    Strefa_3 : DINT  := L#3;
    Strefa_4 : DINT  := L#4;
    Strefa_5 : DINT  := L#4;
    Strefa_6 : DINT  := L#4;
    Strefa_7 : DINT  := L#4;
    Strefa_8 : DINT  := L#4;
    Strefa_9 : DINT  := L#4;
    Strefa_10 : DINT  := L#4;
    Strefa_11 : DINT  := L#4;
    Strefa_12 : DINT  := L#4;
    Strefa_13 : DINT  := L#4;
    Strefa_14 : DINT  := L#4;
    Strefa_15 : DINT  := L#4;
    Strefa_16 : DINT  := L#4;
    Strefa_17 : DINT  := L#4;
    Strefa_18 : DINT  := L#4;
    Strefa_19 : DINT  := L#4;
    Strefa_20 : DINT  := L#4;
    Strefa_21 : DINT  := L#4;
    Strefa_22 : DINT  := L#4;
    Strefa_23 : DINT  := L#4;
    Strefa_24 : DINT  := L#4;
   END_STRUCT ;
   Wartosc_Predkosci : STRUCT 	//Wartosc Predkosci w procentach
    Predkosc_0 : DINT  := L#100;
    Predkosc_1 : DINT  := L#100;
    Predkosc_2 : DINT  := L#100;
    Predkosc_3 : DINT  := L#100;
    Predkosc_4 : DINT  := L#100;
    Predkosc_5 : DINT  := L#100;
    Predkosc_6 : DINT  := L#100;
    Predkosc_7 : DINT  := L#100;
    Predkosc_8 : DINT  := L#100;
    Predkosc_9 : DINT  := L#100;
    Predkosc_10 : DINT  := L#100;
    Predkosc_11 : DINT  := L#100;
    Predkosc_12 : DINT  := L#100;
    Predkosc_13 : DINT  := L#100;
    Predkosc_14 : DINT  := L#100;
    Predkosc_15 : DINT  := L#100;
    Predkosc_16 : DINT  := L#100;
    Predkosc_17 : DINT  := L#100;
    Predkosc_18 : DINT  := L#100;
    Predkosc_19 : DINT  := L#100;
    Predkosc_20 : DINT  := L#100;
    Predkosc_21 : DINT  := L#100;
    Predkosc_22 : DINT  := L#100;
    Predkosc_23 : DINT  := L#100;
    Predkosc_24 : DINT  := L#100;
   END_STRUCT ;
  END_STRUCT ;	
BEGIN
   Wartosc_Pozycji.Poz_1 := L#1000;
   Wartosc_Pozycji.Poz_2 := L#2000;
   Wartosc_Pozycji.Poz_3 := L#5000;
   Wartosc_Pozycji.Poz_4 := L#20000;
   Wartosc_Pozycji.Poz_5 := L#40000;
   Wartosc_Strefy.Strefa_0 := L#4;
   Wartosc_Strefy.Strefa_1 := L#4;
   Wartosc_Strefy.Strefa_2 := L#4;
   Wartosc_Strefy.Strefa_3 := L#4;
   Wartosc_Strefy.Strefa_4 := L#4;
   Wartosc_Strefy.Strefa_5 := L#4;
   Wartosc_Strefy.Strefa_6 := L#4;
   Wartosc_Strefy.Strefa_7 := L#4;
   Wartosc_Strefy.Strefa_8 := L#4;
   Wartosc_Strefy.Strefa_9 := L#4;
   Wartosc_Strefy.Strefa_10 := L#4;
   Wartosc_Strefy.Strefa_11 := L#4;
   Wartosc_Strefy.Strefa_12 := L#4;
   Wartosc_Strefy.Strefa_13 := L#4;
   Wartosc_Strefy.Strefa_14 := L#4;
   Wartosc_Strefy.Strefa_15 := L#4;
   Wartosc_Strefy.Strefa_16 := L#4;
   Wartosc_Strefy.Strefa_17 := L#4;
   Wartosc_Strefy.Strefa_18 := L#4;
   Wartosc_Strefy.Strefa_19 := L#4;
   Wartosc_Strefy.Strefa_20 := L#4;
   Wartosc_Strefy.Strefa_21 := L#4;
   Wartosc_Strefy.Strefa_22 := L#4;
   Wartosc_Strefy.Strefa_23 := L#4;
   Wartosc_Strefy.Strefa_24 := L#4;
   Wartosc_Predkosci.Predkosc_0 := L#100;
   Wartosc_Predkosci.Predkosc_1 := L#100;
   Wartosc_Predkosci.Predkosc_2 := L#100;
   Wartosc_Predkosci.Predkosc_3 := L#100;
   Wartosc_Predkosci.Predkosc_4 := L#100;
   Wartosc_Predkosci.Predkosc_5 := L#100;
   Wartosc_Predkosci.Predkosc_6 := L#100;
   Wartosc_Predkosci.Predkosc_7 := L#100;
   Wartosc_Predkosci.Predkosc_8 := L#100;
   Wartosc_Predkosci.Predkosc_9 := L#100;
   Wartosc_Predkosci.Predkosc_10 := L#100;
   Wartosc_Predkosci.Predkosc_11 := L#100;
   Wartosc_Predkosci.Predkosc_12 := L#100;
   Wartosc_Predkosci.Predkosc_13 := L#100;
   Wartosc_Predkosci.Predkosc_14 := L#100;
   Wartosc_Predkosci.Predkosc_15 := L#100;
   Wartosc_Predkosci.Predkosc_16 := L#100;
   Wartosc_Predkosci.Predkosc_17 := L#100;
   Wartosc_Predkosci.Predkosc_18 := L#100;
   Wartosc_Predkosci.Predkosc_19 := L#100;
   Wartosc_Predkosci.Predkosc_20 := L#100;
   Wartosc_Predkosci.Predkosc_21 := L#100;
   Wartosc_Predkosci.Predkosc_22 := L#100;
   Wartosc_Predkosci.Predkosc_23 := L#100;
   Wartosc_Predkosci.Predkosc_24 := L#100;
END_DATA_BLOCK

DATA_BLOCK "Buffor_Rejestr"	// DB 823
VERSION : 0.1
  STRUCT
   Pozycja_1 : DINT ;	//Pozycja nr 1 na bandzie (wozek)
   Pozycja_2 : DINT ;	//Pozycja nr 2 na bandzie odbierajacej
   Pozycja_3 : DINT ;	//Pozycja nr 3 na bandzie odbierajacej
   Pozycja_4 : DINT ;	//Pozycja nr 4 na bandzie odbierajacej
   Pozycja_5 : DINT ;	//Pozycja nr 5 na bandzie odbierajacej
   Pozycja_6 : DINT ;	//Pozycja nr 6 na bandzie odbierajacej
   Pozycja_rezerwa_7 : DINT ;	//Pozycja rezerwa
   Pozycja_rezerwa_8 : DINT ;	//Pozycja rezerwa
   Pozycja_12 : DINT ;	//Pozycja nr 12
   Pozycja_13 : DINT ;	//Pozycja nr 13
   Pozycja_14 : DINT ;	//Pozycja nr 14
   Pozycja_15 : DINT ;	//Pozycja nr 15
   Pozycja_16 : DINT ;	//Pozycja nr 16
   Pozycja_Shuttle : DINT ;	//Pozycja nr  na bandzie (wozek)
   Pozycja_7 : DINT ;	//Pozycja nr 7
   Pozycja_8 : DINT ;	//Pozycja nr 8
   Pozycja_17 : DINT ;	//Pozycja nr 17
   Pozycja_18 : DINT ;	//Pozycja nr 18
  END_STRUCT ;	
BEGIN
   Pozycja_2 := L#-2147483648;
END_DATA_BLOCK

DATA_BLOCK "Buffor_Rejestr_HMI"	// DB 824
VERSION : 0.1
  STRUCT
   Pozycja_1_HMI : DINT ;	//Pozycja nr 1 na bandzie (wozek)
   Pozycja_2_HMI : DINT ;	//Pozycja nr 2 na bandzie odbierajacej
   Pozycja_3_HMI : DINT ;	//Pozycja nr 3 na bandzie odbierajacej
   Pozycja_4_HMI : DINT ;	//Pozycja nr 4 na bandzie odbierajacej
   Pozycja_5_HMI : DINT ;	//Pozycja nr 5 na bandzie odbierajacej
   Pozycja_6_HMI : DINT ;	//Pozycja nr 6 na bandzie odbierajacej
   Pozycja_rezerwa_7_HMI : DINT ;	//Pozycja rezerwa
   Pozycja_rezerwa_8_HMI : DINT ;	//Pozycja rezerwa
   Pozycja_12_HMI : DINT ;	//Pozycja nr 12
   Pozycja_13_HMI : DINT ;	//Pozycja nr 13
   Pozycja_14_HMI : DINT ;	//Pozycja nr 14
   Pozycja_15_HMI : DINT ;	//Pozycja nr 15
   Pozycja_16_HMI : DINT ;	//Pozycja nr 16
   Pozycja_17_HMI : DINT ;	//Pozycja nr 17 na bandzie (wozek)
  END_STRUCT ;	
BEGIN
   Pozycja_2_HMI := L#-2147483648;
END_DATA_BLOCK

DATA_BLOCK "Def_Stale_Maszynowe"	// DB 830
VERSION : 0.1
  STRUCT
   Pozycja_Skrajna_Dol : DINT  := L#280;
   Pozycja_KB1 : DINT  := L#400;	//Temporary placeholder variable
   Pozycja_KB2 : DINT  := L#15905;
   Pozycja_Gender : DINT  := L#24780;
   Pozycja_odbieranie : DINT  := L#33000;
   Pozycja_Pobieranie : DINT  := L#34180;
   Pozycja_Skrajna_Gora : DINT  := L#34210;
   Reserwa : DINT ;
   War_W_Kolejce_KB1 : DINT  := L#200;
   War_W_Kolejce_KB2 : DINT  := L#200;
   War_W_Kolejce_Intro : DINT  := L#100;
   War_W_Kolejce_Reserwa : DINT ;
   War_W_Kolejce_Reserwa1 : DINT ;
   Reserwa_16 : DINT ;
   Reserwa_20 : DINT ;
   Reserwa_21 : DINT ;
   Reserwa_22 : DINT ;
   Reserwa_24 : DINT ;
   res : DINT ;
   res1 : DINT ;
   res2 : DINT ;
   res3 : DINT ;
   res4 : DINT ;
   res5 : DINT ;
   res6 : DINT ;
   res7 : DINT ;
   res8 : DINT ;
   res81 : DINT ;
   res82 : DINT ;
   res83 : DINT ;
   res84 : DINT ;
   res85 : DINT ;
   res86 : DINT ;
   res87 : DINT ;
   res88 : DINT ;
   res89 : DINT ;
   res810 : DINT ;
   res811 : DINT ;
   res812 : DINT ;
   res813 : DINT ;
   res814 : DINT ;
   res815 : DINT ;
   res816 : DINT ;
   res817 : DINT ;
   res818 : DINT ;
   res819 : DINT ;
   res820 : DINT ;
   res821 : DINT ;
   res822 : DINT ;
   res823 : DINT ;
  END_STRUCT ;	
BEGIN
   Pozycja_Skrajna_Dol := L#280;
   Pozycja_KB1 := L#400;
   Pozycja_KB2 := L#15905;
   Pozycja_Gender := L#24780;
   Pozycja_odbieranie := L#33000;
   Pozycja_Pobieranie := L#34180;
   Pozycja_Skrajna_Gora := L#34210;
   War_W_Kolejce_KB1 := L#200;
   War_W_Kolejce_KB2 := L#200;
   War_W_Kolejce_Intro := L#100;
END_DATA_BLOCK

